LIN {X -190.795,Y +430.646,Z +0.000,A +0.152,E1 -46.707,E3 +41715.361,E4 +0.000} C_DIS
LIN {X -190.395,Y +441.145,Z +0.000,A +0.001,E1 -46.583,E3 +41728.754,E4 +0.000} C_DIS
LIN {X -190.239,Y +451.150,Z +0.000,A -0.000,E1 -46.528,E3 +41741.522,E4 +0.000} C_DIS
LIN {X -190.161,Y +465.026,Z +0.000,A -0.000,E1 -46.506,E3 +41759.237,E4 +0.000} C_DIS
LIN {X -190.142,Y +1057.148,Z +0.000,A -0.000,E1 -46.500,E3 +42515.443,E4 +0.000} C_DIS
LIN {X -190.147,Y +1068.924,Z +0.000,A -0.000,E1 -46.499,E3 +42530.484,E4 +0.000} C_DIS
LIN {X -190.159,Y +1079.072,Z +0.000,A -0.000,E1 -46.493,E3 +42543.449,E4 +0.000} C_DIS
LIN {X -190.174,Y +1086.028,Z +0.000,A -0.000,E1 -46.483,E3 +42552.343,E4 +0.000} C_DIS
LIN {X -190.200,Y +1096.186,Z +0.000,A -0.000,E1 -46.448,E3 +42565.347,E4 +0.000} C_DIS
LIN {X -190.154,Y +1108.998,Z +0.000,A -0.054,E1 -46.295,E3 +42581.842,E4 +0.000} C_DIS
LIN {X -189.772,Y +1119.341,Z +0.000,A -0.752,E1 -45.902,E3 +42595.380,E4 +0.000} C_DIS
LIN {X -189.097,Y +1124.276,Z +0.000,A -2.508,E1 -45.397,E3 +42602.112,E4 +0.000} C_DIS
LIN {X -187.410,Y +1129.069,Z +0.000,A -5.304,E1 -44.585,E3 +42609.285,E4 +0.000} C_DIS
LIN {X -183.899,Y +1134.873,Z +0.000,A -10.372,E1 -42.805,E3 +42619.291,E4 +0.000} C_DIS
LIN {X -179.711,Y +1140.065,Z +0.000,A -15.940,E1 -40.393,E3 +42630.077,E4 +0.000} C_DIS
LIN {X -176.763,Y +1143.197,Z +0.000,A -18.748,E1 -38.674,E3 +42637.815,E4 +0.000} C_DIS
LIN {X -172.185,Y +1147.423,Z +0.000,A -19.971,E1 -36.175,E3 +42650.545,E4 +0.000} C_DIS
LIN {X -165.999,Y +1152.127,Z +0.000,A -20.000,E1 -32.027,E3 +42670.303,E4 +0.000} C_DIS
LIN {X -160.138,Y +1155.667,Z +0.000,A -20.000,E1 -26.368,E3 +42694.673,E4 +0.000} C_DIS
LIN {X -155.625,Y +1157.756,Z +0.000,A -20.000,E1 -19.505,E3 +42723.349,E4 +0.000} C_DIS
LIN {X -153.552,Y +1158.113,Z +0.000,A -20.000,E1 -11.113,E3 +42759.100,E4 +0.000} C_DIS
LIN {X -156.311,Y +1155.540,Z +0.000,A -20.000,E1 -0.839,E3 +42802.460,E4 +0.000} C_DIS
LIN {X -161.281,Y +1151.851,Z +0.000,A -20.000,E1 +7.737,E3 +42832.359,E4 +0.000} C_DIS
LIN {X -167.493,Y +1147.157,Z +0.000,A -20.000,E1 +16.195,E3 +42856.798,E4 +0.000} C_DIS
LIN {X -173.235,Y +1142.221,Z +0.000,A -20.000,E1 +22.930,E3 +42874.100,E4 +0.000} C_DIS
LIN {X -181.123,Y +1133.734,Z +0.000,A -20.000,E1 +30.868,E3 +42894.856,E4 +0.000} C_DIS
LIN {X -189.654,Y +1120.856,Z +0.000,A -20.000,E1 +39.018,E3 +42916.870,E4 +0.000} C_DIS
LIN {X -195.246,Y +1107.046,Z +0.000,A -20.000,E1 +44.515,E3 +42934.772,E4 +0.000} C_DIS
LIN {X -198.051,Y +1092.368,Z +0.000,A -20.000,E1 +47.947,E3 +42951.298,E4 +0.000} C_DIS
LIN {X -198.143,Y +1081.370,Z +0.000,A -19.806,E1 +49.153,E3 +42963.159,E4 +0.000} C_DIS
LIN {X -197.177,Y +1073.569,Z +0.000,A -17.356,E1 +49.162,E3 +42971.743,E4 +0.000} C_DIS
LIN {X -195.448,Y +1066.139,Z +0.000,A -12.154,E1 +48.512,E3 +42980.338,E4 +0.000} C_DIS
LIN {X -193.346,Y +1058.941,Z +0.000,A -7.133,E1 +47.724,E3 +42989.218,E4 +0.000} C_DIS
LIN {X -191.781,Y +1050.839,Z +0.000,A -3.715,E1 +47.274,E3 +42999.551,E4 +0.000} C_DIS
LIN {X -190.795,Y +1039.355,Z +0.000,A -0.983,E1 +46.842,E3 +43014.211,E4 +0.000} C_DIS
LIN {X -190.395,Y +1028.856,Z +0.000,A -0.089,E1 +46.598,E3 +43027.605,E4 +0.000} C_DIS
LIN {X -190.239,Y +1018.851,Z +0.000,A -0.004,E1 +46.529,E3 +43040.373,E4 +0.000} C_DIS
LIN {X -190.161,Y +1004.975,Z +0.000,A +0.000,E1 +46.506,E3 +43058.087,E4 +0.000} C_DIS
LIN {X -190.142,Y +412.853,Z +0.000,A +0.000,E1 +46.501,E3 +43814.293,E4 +0.000} C_DIS
LIN {X -190.147,Y +401.077,Z +0.000,A +0.000,E1 +46.499,E3 +43829.334,E4 +0.000} C_DIS
LIN {X -190.159,Y +390.929,Z +0.000,A +0.000,E1 +46.494,E3 +43842.300,E4 +0.000} C_DIS
LIN {X -190.174,Y +383.973,Z +0.000,A +0.000,E1 +46.484,E3 +43851.193,E4 +0.000} C_DIS
LIN {X -190.200,Y +373.815,Z +0.000,A +0.000,E1 +46.448,E3 +43864.198,E4 +0.000} C_DIS
LIN {X -190.154,Y +361.003,Z +0.000,A +0.000,E1 +46.303,E3 +43880.692,E4 +0.000} C_DIS
LIN {X -189.772,Y +350.660,Z +0.000,A +0.049,E1 +45.996,E3 +43894.231,E4 +0.000} C_DIS
LIN {X -189.325,Y +346.917,Z +0.000,A +0.243,E1 +45.771,E3 +43899.300,E4 +0.000} C_DIS
LIN {X -188.196,Y +342.754,Z +0.000,A +1.966,E1 +45.249,E3 +43905.308,E4 +0.000} C_DIS
LIN {X -185.199,Y +337.023,Z +0.000,A +6.630,E1 +43.793,E3 +43914.682,E4 +0.000} C_DIS
LIN {X -181.141,Y +331.596,Z +0.000,A +12.274,E1 +41.569,E3 +43925.242,E4 +0.000} C_DIS
LIN {X -176.762,Y +326.804,Z +0.000,A +17.560,E1 +38.898,E3 +43936.666,E4 +0.000} C_DIS
LIN {X -172.184,Y +322.578,Z +0.000,A +19.859,E1 +36.197,E3 +43949.396,E4 +0.000} C_DIS
LIN {X -165.998,Y +317.874,Z +0.000,A +20.000,E1 +32.027,E3 +43969.154,E4 +0.000} C_DIS
LIN {X -160.137,Y +314.334,Z +0.000,A +20.000,E1 +26.368,E3 +43993.523,E4 +0.000} C_DIS
LIN {X -155.624,Y +312.245,Z +0.000,A +20.000,E1 +19.506,E3 +44022.199,E4 +0.000} C_DIS
LIN {X -153.557,Y +311.879,Z +0.000,A +20.000,E1 +11.113,E3 +44057.954,E4 +0.000} C_DIS
LIN {X -155.320,Y +313.348,Z +0.000,A +20.000,E1 +3.401,E3 +44091.138,E4 +0.000} C_DIS
LIN {X -160.005,Y +315.804,Z +0.000,A +20.000,E1 -4.720,E3 +44121.516,E4 +0.000} C_DIS
LIN {X -164.504,Y +318.255,Z +0.000,A +20.000,E1 -10.663,E3 +44140.885,E4 +0.000} C_DIS
LIN {X -170.340,Y +322.684,Z +0.000,A +20.000,E1 -17.457,E3 +44160.917,E4 +0.000} C_DIS
LIN {X -175.568,Y +329.106,Z +0.000,A +20.000,E1 -24.747,E3 +44178.151,E4 +0.000} C_DIS
LIN {X -184.074,Y +340.065,Z +0.000,A +20.000,E1 -33.664,E3 +44201.091,E4 +0.000} C_DIS
LIN {X -190.779,Y +351.388,Z +0.000,A +20.000,E1 -40.083,E3 +44218.869,E4 +0.000} C_DIS
LIN {X -195.254,Y +362.955,Z +0.000,A +20.000,E1 -44.515,E3 +44233.622,E4 +0.000} C_DIS
LIN {X -197.754,Y +374.780,Z +0.000,A +20.000,E1 -47.450,E3 +44247.044,E4 +0.000} C_DIS
LIN {X -198.310,Y +383.215,Z +0.000,A +19.956,E1 -48.698,E3 +44256.168,E4 +0.000} C_DIS
LIN {X -197.912,Y +391.275,Z +0.000,A +18.601,E1 -49.158,E3 +44264.886,E4 +0.000} C_DIS
LIN {X -196.679,Y +398.944,Z +0.000,A +13.989,E1 -48.784,E3 +44273.440,E4 +0.000} C_DIS
LIN {X -194.742,Y +406.288,Z +0.000,A +8.476,E1 -48.001,E3 +44282.123,E4 +0.000} C_DIS
LIN {X -192.748,Y +413.472,Z +0.000,A +3.905,E1 -47.267,E3 +44291.133,E4 +0.000} C_DIS
LIN {X -191.781,Y +419.162,Z +0.000,A +1.739,E1 -46.975,E3 +44298.401,E4 +0.000} C_DIS
LIN {X -190.795,Y +430.646,Z +0.000,A +0.152,E1 -46.707,E3 +44313.062,E4 +0.000} C_DIS
LIN {X -190.395,Y +441.145,Z +0.000,A +0.001,E1 -46.583,E3 +44326.455,E4 +0.000} C_DIS
LIN {X -190.239,Y +451.150,Z +0.000,A -0.000,E1 -46.528,E3 +44339.223,E4 +0.000} C_DIS
LIN {X -190.161,Y +465.026,Z +0.000,A -0.000,E1 -46.506,E3 +44356.938,E4 +0.000} C_DIS
LIN {X -190.142,Y +1057.148,Z +0.000,A -0.000,E1 -46.500,E3 +45113.144,E4 +0.000} C_DIS
LIN {X -190.147,Y +1068.924,Z +0.000,A -0.000,E1 -46.499,E3 +45128.185,E4 +0.000} C_DIS
LIN {X -190.159,Y +1079.072,Z +0.000,A -0.000,E1 -46.493,E3 +45141.150,E4 +0.000} C_DIS
LIN {X -190.174,Y +1086.028,Z +0.000,A -0.000,E1 -46.483,E3 +45150.044,E4 +0.000} C_DIS
LIN {X -190.200,Y +1096.186,Z +0.000,A -0.000,E1 -46.448,E3 +45163.048,E4 +0.000} C_DIS
LIN {X -190.154,Y +1108.998,Z +0.000,A -0.054,E1 -46.295,E3 +45179.543,E4 +0.000} C_DIS
LIN {X -189.772,Y +1119.341,Z +0.000,A -0.752,E1 -45.902,E3 +45193.081,E4 +0.000} C_DIS
LIN {X -189.097,Y +1124.276,Z +0.000,A -2.508,E1 -45.397,E3 +45199.813,E4 +0.000} C_DIS
LIN {X -187.410,Y +1129.069,Z +0.000,A -5.304,E1 -44.585,E3 +45206.986,E4 +0.000} C_DIS
LIN {X -183.899,Y +1134.873,Z +0.000,A -10.372,E1 -42.805,E3 +45216.992,E4 +0.000} C_DIS
LIN {X -179.711,Y +1140.065,Z +0.000,A -15.940,E1 -40.393,E3 +45227.778,E4 +0.000} C_DIS
LIN {X -176.763,Y +1143.197,Z +0.000,A -18.748,E1 -38.674,E3 +45235.516,E4 +0.000} C_DIS
LIN {X -172.185,Y +1147.423,Z +0.000,A -19.971,E1 -36.175,E3 +45248.246,E4 +0.000} C_DIS
LIN {X -165.999,Y +1152.127,Z +0.000,A -20.000,E1 -32.027,E3 +45268.004,E4 +0.000} C_DIS
LIN {X -160.138,Y +1155.667,Z +0.000,A -20.000,E1 -26.368,E3 +45292.374,E4 +0.000} C_DIS
LIN {X -155.625,Y +1157.756,Z +0.000,A -20.000,E1 -19.505,E3 +45321.050,E4 +0.000} C_DIS
LIN {X -153.552,Y +1158.113,Z +0.000,A -20.000,E1 -11.113,E3 +45356.801,E4 +0.000} C_DIS
LIN {X -156.311,Y +1155.540,Z +0.000,A -20.000,E1 -0.839,E3 +45400.161,E4 +0.000} C_DIS
LIN {X -161.281,Y +1151.851,Z +0.000,A -20.000,E1 +7.737,E3 +45430.060,E4 +0.000} C_DIS
LIN {X -167.493,Y +1147.157,Z +0.000,A -20.000,E1 +16.195,E3 +45454.499,E4 +0.000} C_DIS
LIN {X -173.235,Y +1142.221,Z +0.000,A -20.000,E1 +22.930,E3 +45471.801,E4 +0.000} C_DIS
LIN {X -181.123,Y +1133.734,Z +0.000,A -20.000,E1 +30.868,E3 +45492.557,E4 +0.000} C_DIS
LIN {X -189.654,Y +1120.856,Z +0.000,A -20.000,E1 +39.018,E3 +45514.571,E4 +0.000} C_DIS
LIN {X -195.246,Y +1107.046,Z +0.000,A -20.000,E1 +44.515,E3 +45532.473,E4 +0.000} C_DIS
LIN {X -198.051,Y +1092.368,Z +0.000,A -20.000,E1 +47.947,E3 +45548.999,E4 +0.000} C_DIS
LIN {X -198.143,Y +1081.370,Z +0.000,A -19.806,E1 +49.153,E3 +45560.860,E4 +0.000} C_DIS
LIN {X -197.177,Y +1073.569,Z +0.000,A -17.356,E1 +49.162,E3 +45569.444,E4 +0.000} C_DIS
LIN {X -195.448,Y +1066.139,Z +0.000,A -12.154,E1 +48.512,E3 +45578.039,E4 +0.000} C_DIS
LIN {X -193.346,Y +1058.941,Z +0.000,A -7.133,E1 +47.724,E3 +45586.919,E4 +0.000} C_DIS
LIN {X -191.781,Y +1050.839,Z +0.000,A -3.715,E1 +47.274,E3 +45597.252,E4 +0.000} C_DIS
LIN {X -190.795,Y +1039.355,Z +0.000,A -0.983,E1 +46.842,E3 +45611.912,E4 +0.000} C_DIS
LIN {X -190.395,Y +1028.856,Z +0.000,A -0.089,E1 +46.598,E3 +45625.306,E4 +0.000} C_DIS
LIN {X -190.239,Y +1018.851,Z +0.000,A -0.004,E1 +46.529,E3 +45638.074,E4 +0.000} C_DIS
LIN {X -190.161,Y +1004.975,Z +0.000,A +0.000,E1 +46.506,E3 +45655.788,E4 +0.000} C_DIS
LIN {X -190.142,Y +412.853,Z +0.000,A +0.000,E1 +46.501,E3 +46411.994,E4 +0.000} C_DIS
LIN {X -190.147,Y +401.077,Z +0.000,A +0.000,E1 +46.499,E3 +46427.035,E4 +0.000} C_DIS
LIN {X -190.159,Y +390.929,Z +0.000,A +0.000,E1 +46.494,E3 +46440.001,E4 +0.000} C_DIS
LIN {X -190.174,Y +383.973,Z +0.000,A +0.000,E1 +46.484,E3 +46448.894,E4 +0.000} C_DIS
LIN {X -190.200,Y +373.815,Z +0.000,A +0.000,E1 +46.448,E3 +46461.899,E4 +0.000} C_DIS
LIN {X -190.154,Y +361.003,Z +0.000,A +0.000,E1 +46.303,E3 +46478.393,E4 +0.000} C_DIS
LIN {X -189.772,Y +350.660,Z +0.000,A +0.049,E1 +45.996,E3 +46491.932,E4 +0.000} C_DIS
LIN {X -189.325,Y +346.917,Z +0.000,A +0.243,E1 +45.771,E3 +46497.001,E4 +0.000} C_DIS
LIN {X -188.196,Y +342.754,Z +0.000,A +1.966,E1 +45.249,E3 +46503.009,E4 +0.000} C_DIS
LIN {X -185.199,Y +337.023,Z +0.000,A +6.630,E1 +43.793,E3 +46512.383,E4 +0.000} C_DIS
LIN {X -181.141,Y +331.596,Z +0.000,A +12.274,E1 +41.569,E3 +46522.943,E4 +0.000} C_DIS
LIN {X -176.762,Y +326.804,Z +0.000,A +17.560,E1 +38.898,E3 +46534.367,E4 +0.000} C_DIS
LIN {X -172.184,Y +322.578,Z +0.000,A +19.859,E1 +36.197,E3 +46547.097,E4 +0.000} C_DIS
LIN {X -165.998,Y +317.874,Z +0.000,A +20.000,E1 +32.027,E3 +46566.855,E4 +0.000} C_DIS
LIN {X -160.137,Y +314.334,Z +0.000,A +20.000,E1 +26.368,E3 +46591.224,E4 +0.000} C_DIS
LIN {X -155.624,Y +312.245,Z +0.000,A +20.000,E1 +19.506,E3 +46619.900,E4 +0.000} C_DIS
LIN {X -153.557,Y +311.879,Z +0.000,A +20.000,E1 +11.113,E3 +46655.655,E4 +0.000} C_DIS
LIN {X -155.320,Y +313.348,Z +0.000,A +20.000,E1 +3.401,E3 +46688.839,E4 +0.000} C_DIS
LIN {X -160.005,Y +315.804,Z +0.000,A +20.000,E1 -4.720,E3 +46719.217,E4 +0.000} C_DIS
LIN {X -164.504,Y +318.255,Z +0.000,A +20.000,E1 -10.663,E3 +46738.586,E4 +0.000} C_DIS
LIN {X -170.340,Y +322.684,Z +0.000,A +20.000,E1 -17.457,E3 +46758.618,E4 +0.000} C_DIS
LIN {X -175.568,Y +329.106,Z +0.000,A +20.000,E1 -24.747,E3 +46775.852,E4 +0.000} C_DIS
LIN {X -184.074,Y +340.065,Z +0.000,A +20.000,E1 -33.664,E3 +46798.792,E4 +0.000} C_DIS
LIN {X -190.779,Y +351.388,Z +0.000,A +20.000,E1 -40.083,E3 +46816.570,E4 +0.000} C_DIS
LIN {X -195.254,Y +362.955,Z +0.000,A +20.000,E1 -44.515,E3 +46831.323,E4 +0.000} C_DIS
LIN {X -197.754,Y +374.780,Z +0.000,A +20.000,E1 -47.450,E3 +46844.745,E4 +0.000} C_DIS
LIN {X -198.310,Y +383.215,Z +0.000,A +19.956,E1 -48.698,E3 +46853.869,E4 +0.000} C_DIS
LIN {X -197.912,Y +391.275,Z +0.000,A +18.601,E1 -49.158,E3 +46862.587,E4 +0.000} C_DIS
LIN {X -196.679,Y +398.944,Z +0.000,A +13.989,E1 -48.784,E3 +46871.141,E4 +0.000} C_DIS
LIN {X -194.742,Y +406.288,Z +0.000,A +8.476,E1 -48.001,E3 +46879.824,E4 +0.000} C_DIS
LIN {X -192.748,Y +413.472,Z +0.000,A +3.905,E1 -47.267,E3 +46888.834,E4 +0.000} C_DIS
LIN {X -191.781,Y +419.162,Z +0.000,A +1.739,E1 -46.975,E3 +46896.102,E4 +0.000} C_DIS
LIN {X -190.795,Y +430.646,Z +0.000,A +0.152,E1 -46.707,E3 +46910.763,E4 +0.000} C_DIS
LIN {X -190.395,Y +441.145,Z +0.000,A +0.001,E1 -46.583,E3 +46924.156,E4 +0.000} C_DIS
LIN {X -190.239,Y +451.150,Z +0.000,A -0.000,E1 -46.528,E3 +46936.924,E4 +0.000} C_DIS
LIN {X -190.161,Y +465.026,Z +0.000,A -0.000,E1 -46.506,E3 +46954.639,E4 +0.000} C_DIS
LIN {X -190.142,Y +1057.148,Z +0.000,A -0.000,E1 -46.500,E3 +47710.845,E4 +0.000} C_DIS
LIN {X -190.147,Y +1068.924,Z +0.000,A -0.000,E1 -46.499,E3 +47725.886,E4 +0.000} C_DIS
LIN {X -190.159,Y +1079.072,Z +0.000,A -0.000,E1 -46.493,E3 +47738.851,E4 +0.000} C_DIS
LIN {X -190.174,Y +1086.028,Z +0.000,A -0.000,E1 -46.483,E3 +47747.745,E4 +0.000} C_DIS
LIN {X -190.200,Y +1096.186,Z +0.000,A -0.000,E1 -46.448,E3 +47760.749,E4 +0.000} C_DIS
LIN {X -190.154,Y +1108.998,Z +0.000,A -0.054,E1 -46.295,E3 +47777.244,E4 +0.000} C_DIS
LIN {X -189.772,Y +1119.341,Z +0.000,A -0.752,E1 -45.902,E3 +47790.782,E4 +0.000} C_DIS
LIN {X -189.097,Y +1124.276,Z +0.000,A -2.508,E1 -45.397,E3 +47797.514,E4 +0.000} C_DIS
LIN {X -187.410,Y +1129.069,Z +0.000,A -5.304,E1 -44.585,E3 +47804.687,E4 +0.000} C_DIS
LIN {X -183.899,Y +1134.873,Z +0.000,A -10.372,E1 -42.805,E3 +47814.693,E4 +0.000} C_DIS
LIN {X -179.711,Y +1140.065,Z +0.000,A -15.940,E1 -40.393,E3 +47825.479,E4 +0.000} C_DIS
LIN {X -176.763,Y +1143.197,Z +0.000,A -18.748,E1 -38.674,E3 +47833.217,E4 +0.000} C_DIS
LIN {X -172.185,Y +1147.423,Z +0.000,A -19.971,E1 -36.175,E3 +47845.947,E4 +0.000} C_DIS
LIN {X -165.999,Y +1152.127,Z +0.000,A -20.000,E1 -32.027,E3 +47865.705,E4 +0.000} C_DIS
LIN {X -160.138,Y +1155.667,Z +0.000,A -20.000,E1 -26.368,E3 +47890.075,E4 +0.000} C_DIS
LIN {X -155.625,Y +1157.756,Z +0.000,A -20.000,E1 -19.505,E3 +47918.751,E4 +0.000} C_DIS
LIN {X -153.552,Y +1158.113,Z +0.000,A -20.000,E1 -11.113,E3 +47954.502,E4 +0.000} C_DIS
LIN {X -156.311,Y +1155.540,Z +0.000,A -20.000,E1 -0.839,E3 +47997.862,E4 +0.000} C_DIS
LIN {X -161.281,Y +1151.851,Z +0.000,A -20.000,E1 +7.737,E3 +48027.761,E4 +0.000} C_DIS
LIN {X -167.493,Y +1147.157,Z +0.000,A -20.000,E1 +16.195,E3 +48052.200,E4 +0.000} C_DIS
LIN {X -173.235,Y +1142.221,Z +0.000,A -20.000,E1 +22.930,E3 +48069.502,E4 +0.000} C_DIS
LIN {X -181.123,Y +1133.734,Z +0.000,A -20.000,E1 +30.868,E3 +48090.258,E4 +0.000} C_DIS
LIN {X -189.654,Y +1120.856,Z +0.000,A -20.000,E1 +39.018,E3 +48112.272,E4 +0.000} C_DIS
LIN {X -195.246,Y +1107.046,Z +0.000,A -20.000,E1 +44.515,E3 +48130.174,E4 +0.000} C_DIS
LIN {X -198.051,Y +1092.368,Z +0.000,A -20.000,E1 +47.947,E3 +48146.700,E4 +0.000} C_DIS
LIN {X -198.143,Y +1081.370,Z +0.000,A -19.806,E1 +49.153,E3 +48158.561,E4 +0.000} C_DIS
LIN {X -197.177,Y +1073.569,Z +0.000,A -17.356,E1 +49.162,E3 +48167.145,E4 +0.000} C_DIS
LIN {X -195.448,Y +1066.139,Z +0.000,A -12.154,E1 +48.512,E3 +48175.740,E4 +0.000} C_DIS
LIN {X -193.346,Y +1058.941,Z +0.000,A -7.133,E1 +47.724,E3 +48184.620,E4 +0.000} C_DIS
LIN {X -191.781,Y +1050.839,Z +0.000,A -3.715,E1 +47.274,E3 +48194.953,E4 +0.000} C_DIS
LIN {X -190.795,Y +1039.355,Z +0.000,A -0.983,E1 +46.842,E3 +48209.613,E4 +0.000} C_DIS
LIN {X -190.395,Y +1028.856,Z +0.000,A -0.089,E1 +46.598,E3 +48223.007,E4 +0.000} C_DIS
LIN {X -190.239,Y +1018.851,Z +0.000,A -0.004,E1 +46.529,E3 +48235.775,E4 +0.000} C_DIS
LIN {X -190.161,Y +1004.975,Z +0.000,A +0.000,E1 +46.506,E3 +48253.489,E4 +0.000} C_DIS
LIN {X -190.142,Y +412.853,Z +0.000,A +0.000,E1 +46.501,E3 +49009.695,E4 +0.000} C_DIS
LIN {X -190.147,Y +401.077,Z +0.000,A +0.000,E1 +46.499,E3 +49024.736,E4 +0.000} C_DIS
LIN {X -190.159,Y +390.929,Z +0.000,A +0.000,E1 +46.494,E3 +49037.702,E4 +0.000} C_DIS
LIN {X -190.174,Y +383.973,Z +0.000,A +0.000,E1 +46.484,E3 +49046.595,E4 +0.000} C_DIS
LIN {X -190.200,Y +373.815,Z +0.000,A +0.000,E1 +46.448,E3 +49059.600,E4 +0.000} C_DIS
LIN {X -190.154,Y +361.003,Z +0.000,A +0.000,E1 +46.303,E3 +49076.094,E4 +0.000} C_DIS
LIN {X -189.772,Y +350.660,Z +0.000,A +0.049,E1 +45.996,E3 +49089.633,E4 +0.000} C_DIS
LIN {X -189.325,Y +346.917,Z +0.000,A +0.243,E1 +45.771,E3 +49094.702,E4 +0.000} C_DIS
LIN {X -188.196,Y +342.754,Z +0.000,A +1.966,E1 +45.249,E3 +49100.710,E4 +0.000} C_DIS
LIN {X -185.199,Y +337.023,Z +0.000,A +6.630,E1 +43.793,E3 +49110.084,E4 +0.000} C_DIS
LIN {X -181.141,Y +331.596,Z +0.000,A +12.274,E1 +41.569,E3 +49120.644,E4 +0.000} C_DIS
LIN {X -176.762,Y +326.804,Z +0.000,A +17.560,E1 +38.898,E3 +49132.068,E4 +0.000} C_DIS
LIN {X -172.184,Y +322.578,Z +0.000,A +19.859,E1 +36.197,E3 +49144.798,E4 +0.000} C_DIS
LIN {X -165.998,Y +317.874,Z +0.000,A +20.000,E1 +32.027,E3 +49164.556,E4 +0.000} C_DIS
LIN {X -160.137,Y +314.334,Z +0.000,A +20.000,E1 +26.368,E3 +49188.925,E4 +0.000} C_DIS
LIN {X -155.624,Y +312.245,Z +0.000,A +20.000,E1 +19.506,E3 +49217.601,E4 +0.000} C_DIS
LIN {X -153.557,Y +311.879,Z +0.000,A +20.000,E1 +11.113,E3 +49253.356,E4 +0.000} C_DIS
LIN {X -155.320,Y +313.348,Z +0.000,A +20.000,E1 +3.401,E3 +49286.540,E4 +0.000} C_DIS
LIN {X -160.005,Y +315.804,Z +0.000,A +20.000,E1 -4.720,E3 +49316.918,E4 +0.000} C_DIS
LIN {X -164.504,Y +318.255,Z +0.000,A +20.000,E1 -10.663,E3 +49336.287,E4 +0.000} C_DIS
LIN {X -170.340,Y +322.684,Z +0.000,A +20.000,E1 -17.457,E3 +49356.319,E4 +0.000} C_DIS
LIN {X -175.568,Y +329.106,Z +0.000,A +20.000,E1 -24.747,E3 +49373.553,E4 +0.000} C_DIS
LIN {X -184.074,Y +340.065,Z +0.000,A +20.000,E1 -33.664,E3 +49396.493,E4 +0.000} C_DIS
LIN {X -190.779,Y +351.388,Z +0.000,A +20.000,E1 -40.083,E3 +49414.271,E4 +0.000} C_DIS
LIN {X -195.254,Y +362.955,Z +0.000,A +20.000,E1 -44.515,E3 +49429.024,E4 +0.000} C_DIS
LIN {X -197.754,Y +374.780,Z +0.000,A +20.000,E1 -47.450,E3 +49442.446,E4 +0.000} C_DIS
LIN {X -198.310,Y +383.215,Z +0.000,A +19.956,E1 -48.698,E3 +49451.570,E4 +0.000} C_DIS
LIN {X -197.912,Y +391.275,Z +0.000,A +18.601,E1 -49.158,E3 +49460.288,E4 +0.000} C_DIS
LIN {X -196.679,Y +398.944,Z +0.000,A +13.989,E1 -48.784,E3 +49468.842,E4 +0.000} C_DIS
LIN {X -194.742,Y +406.288,Z +0.000,A +8.476,E1 -48.001,E3 +49477.525,E4 +0.000} C_DIS
LIN {X -192.748,Y +413.472,Z +0.000,A +3.905,E1 -47.267,E3 +49486.535,E4 +0.000} C_DIS
LIN {X -191.781,Y +419.162,Z +0.000,A +1.739,E1 -46.975,E3 +49493.803,E4 +0.000} C_DIS
LIN {X -190.795,Y +430.646,Z +0.000,A +0.152,E1 -46.707,E3 +49508.464,E4 +0.000} C_DIS
LIN {X -190.395,Y +441.145,Z +0.000,A +0.001,E1 -46.583,E3 +49521.857,E4 +0.000} C_DIS
LIN {X -190.239,Y +451.150,Z +0.000,A -0.000,E1 -46.528,E3 +49534.625,E4 +0.000} C_DIS
LIN {X -190.161,Y +465.026,Z +0.000,A -0.000,E1 -46.506,E3 +49552.340,E4 +0.000} C_DIS
LIN {X -190.142,Y +1057.148,Z +0.000,A -0.000,E1 -46.500,E3 +50308.546,E4 +0.000} C_DIS
LIN {X -190.147,Y +1068.924,Z +0.000,A -0.000,E1 -46.499,E3 +50323.587,E4 +0.000} C_DIS
LIN {X -190.159,Y +1079.072,Z +0.000,A -0.000,E1 -46.493,E3 +50336.552,E4 +0.000} C_DIS
LIN {X -190.174,Y +1086.028,Z +0.000,A -0.000,E1 -46.483,E3 +50345.446,E4 +0.000} C_DIS
LIN {X -190.200,Y +1096.186,Z +0.000,A -0.000,E1 -46.448,E3 +50358.450,E4 +0.000} C_DIS
LIN {X -190.154,Y +1108.998,Z +0.000,A -0.054,E1 -46.295,E3 +50374.945,E4 +0.000} C_DIS
LIN {X -189.772,Y +1119.341,Z +0.000,A -0.752,E1 -45.902,E3 +50388.483,E4 +0.000} C_DIS
LIN {X -189.097,Y +1124.276,Z +0.000,A -2.508,E1 -45.397,E3 +50395.215,E4 +0.000} C_DIS
LIN {X -187.410,Y +1129.069,Z +0.000,A -5.304,E1 -44.585,E3 +50402.388,E4 +0.000} C_DIS
LIN {X -183.899,Y +1134.873,Z +0.000,A -10.372,E1 -42.805,E3 +50412.394,E4 +0.000} C_DIS
LIN {X -179.711,Y +1140.065,Z +0.000,A -15.940,E1 -40.393,E3 +50423.180,E4 +0.000} C_DIS
LIN {X -176.763,Y +1143.197,Z +0.000,A -18.748,E1 -38.674,E3 +50430.918,E4 +0.000} C_DIS
LIN {X -172.185,Y +1147.423,Z +0.000,A -19.971,E1 -36.175,E3 +50443.648,E4 +0.000} C_DIS
LIN {X -165.999,Y +1152.127,Z +0.000,A -20.000,E1 -32.027,E3 +50463.406,E4 +0.000} C_DIS
LIN {X -160.138,Y +1155.667,Z +0.000,A -20.000,E1 -26.368,E3 +50487.776,E4 +0.000} C_DIS
LIN {X -155.625,Y +1157.756,Z +0.000,A -20.000,E1 -19.505,E3 +50516.452,E4 +0.000} C_DIS
LIN {X -153.552,Y +1158.113,Z +0.000,A -20.000,E1 -11.113,E3 +50552.203,E4 +0.000} C_DIS
LIN {X -156.311,Y +1155.540,Z +0.000,A -20.000,E1 -0.839,E3 +50595.563,E4 +0.000} C_DIS
LIN {X -161.281,Y +1151.851,Z +0.000,A -20.000,E1 +7.737,E3 +50625.462,E4 +0.000} C_DIS
LIN {X -167.493,Y +1147.157,Z +0.000,A -20.000,E1 +16.195,E3 +50649.901,E4 +0.000} C_DIS
LIN {X -173.235,Y +1142.221,Z +0.000,A -20.000,E1 +22.930,E3 +50667.203,E4 +0.000} C_DIS
LIN {X -181.123,Y +1133.734,Z +0.000,A -20.000,E1 +30.868,E3 +50687.959,E4 +0.000} C_DIS
LIN {X -189.654,Y +1120.856,Z +0.000,A -20.000,E1 +39.018,E3 +50709.973,E4 +0.000} C_DIS
LIN {X -195.246,Y +1107.046,Z +0.000,A -20.000,E1 +44.515,E3 +50727.875,E4 +0.000} C_DIS
LIN {X -198.051,Y +1092.368,Z +0.000,A -20.000,E1 +47.947,E3 +50744.401,E4 +0.000} C_DIS
LIN {X -198.143,Y +1081.370,Z +0.000,A -19.806,E1 +49.153,E3 +50756.262,E4 +0.000} C_DIS
LIN {X -197.177,Y +1073.569,Z +0.000,A -17.356,E1 +49.162,E3 +50764.846,E4 +0.000} C_DIS
LIN {X -195.448,Y +1066.139,Z +0.000,A -12.154,E1 +48.512,E3 +50773.441,E4 +0.000} C_DIS
LIN {X -193.346,Y +1058.941,Z +0.000,A -7.133,E1 +47.724,E3 +50782.321,E4 +0.000} C_DIS
LIN {X -191.781,Y +1050.839,Z +0.000,A -3.715,E1 +47.274,E3 +50792.654,E4 +0.000} C_DIS
LIN {X -190.795,Y +1039.355,Z +0.000,A -0.983,E1 +46.842,E3 +50807.314,E4 +0.000} C_DIS
LIN {X -190.395,Y +1028.856,Z +0.000,A -0.089,E1 +46.598,E3 +50820.708,E4 +0.000} C_DIS
LIN {X -190.239,Y +1018.851,Z +0.000,A -0.004,E1 +46.529,E3 +50833.476,E4 +0.000} C_DIS
LIN {X -190.161,Y +1004.975,Z +0.000,A +0.000,E1 +46.506,E3 +50851.190,E4 +0.000} C_DIS
LIN {X -190.142,Y +412.853,Z +0.000,A +0.000,E1 +46.501,E3 +51607.396,E4 +0.000} C_DIS
LIN {X -190.147,Y +401.077,Z +0.000,A +0.000,E1 +46.499,E3 +51622.437,E4 +0.000} C_DIS
LIN {X -190.159,Y +390.929,Z +0.000,A +0.000,E1 +46.494,E3 +51635.403,E4 +0.000} C_DIS
LIN {X -190.174,Y +383.973,Z +0.000,A +0.000,E1 +46.484,E3 +51644.296,E4 +0.000} C_DIS
LIN {X -190.200,Y +373.815,Z +0.000,A +0.000,E1 +46.448,E3 +51657.301,E4 +0.000} C_DIS
LIN {X -190.154,Y +361.003,Z +0.000,A +0.000,E1 +46.303,E3 +51673.795,E4 +0.000} C_DIS
LIN {X -189.772,Y +350.660,Z +0.000,A +0.049,E1 +45.996,E3 +51687.334,E4 +0.000} C_DIS
LIN {X -189.325,Y +346.917,Z +0.000,A +0.243,E1 +45.771,E3 +51692.403,E4 +0.000} C_DIS
LIN {X -188.196,Y +342.754,Z +0.000,A +1.966,E1 +45.249,E3 +51698.411,E4 +0.000} C_DIS
LIN {X -185.199,Y +337.023,Z +0.000,A +6.630,E1 +43.793,E3 +51707.785,E4 +0.000} C_DIS
LIN {X -181.141,Y +331.596,Z +0.000,A +12.274,E1 +41.569,E3 +51718.345,E4 +0.000} C_DIS
LIN {X -176.762,Y +326.804,Z +0.000,A +17.560,E1 +38.898,E3 +51729.769,E4 +0.000} C_DIS
LIN {X -172.184,Y +322.578,Z +0.000,A +19.859,E1 +36.197,E3 +51742.499,E4 +0.000} C_DIS
LIN {X -165.998,Y +317.874,Z +0.000,A +20.000,E1 +32.027,E3 +51762.257,E4 +0.000} C_DIS
LIN {X -160.137,Y +314.334,Z +0.000,A +20.000,E1 +26.368,E3 +51786.626,E4 +0.000} C_DIS
LIN {X -155.624,Y +312.245,Z +0.000,A +20.000,E1 +19.506,E3 +51815.302,E4 +0.000} C_DIS
LIN {X -153.557,Y +311.879,Z +0.000,A +20.000,E1 +11.113,E3 +51851.057,E4 +0.000} C_DIS
LIN {X -155.320,Y +313.348,Z +0.000,A +20.000,E1 +3.401,E3 +51884.241,E4 +0.000} C_DIS
LIN {X -160.005,Y +315.804,Z +0.000,A +20.000,E1 -4.720,E3 +51914.619,E4 +0.000} C_DIS
LIN {X -164.504,Y +318.255,Z +0.000,A +20.000,E1 -10.663,E3 +51933.988,E4 +0.000} C_DIS
LIN {X -170.340,Y +322.684,Z +0.000,A +20.000,E1 -17.457,E3 +51954.020,E4 +0.000} C_DIS
LIN {X -175.568,Y +329.106,Z +0.000,A +20.000,E1 -24.747,E3 +51971.254,E4 +0.000} C_DIS
LIN {X -184.074,Y +340.065,Z +0.000,A +20.000,E1 -33.664,E3 +51994.194,E4 +0.000} C_DIS
LIN {X -190.779,Y +351.388,Z +0.000,A +20.000,E1 -40.083,E3 +52011.972,E4 +0.000} C_DIS
LIN {X -195.254,Y +362.955,Z +0.000,A +20.000,E1 -44.515,E3 +52026.725,E4 +0.000} C_DIS
LIN {X -197.754,Y +374.780,Z +0.000,A +20.000,E1 -47.450,E3 +52040.147,E4 +0.000} C_DIS
LIN {X -198.310,Y +383.215,Z +0.000,A +19.956,E1 -48.698,E3 +52049.271,E4 +0.000} C_DIS
LIN {X -197.912,Y +391.275,Z +0.000,A +18.601,E1 -49.158,E3 +52057.989,E4 +0.000} C_DIS
LIN {X -196.679,Y +398.944,Z +0.000,A +13.989,E1 -48.784,E3 +52066.543,E4 +0.000} C_DIS
LIN {X -194.742,Y +406.288,Z +0.000,A +8.476,E1 -48.001,E3 +52075.226,E4 +0.000} C_DIS
LIN {X -192.748,Y +413.472,Z +0.000,A +3.905,E1 -47.267,E3 +52084.236,E4 +0.000} C_DIS
LIN {X -191.781,Y +419.162,Z +0.000,A +1.739,E1 -46.975,E3 +52091.504,E4 +0.000} C_DIS
LIN {X -190.795,Y +430.646,Z +0.000,A +0.152,E1 -46.707,E3 +52106.165,E4 +0.000} C_DIS
LIN {X -190.395,Y +441.145,Z +0.000,A +0.001,E1 -46.583,E3 +52119.558,E4 +0.000} C_DIS
LIN {X -190.239,Y +451.150,Z +0.000,A -0.000,E1 -46.528,E3 +52132.326,E4 +0.000} C_DIS
LIN {X -190.161,Y +465.026,Z +0.000,A -0.000,E1 -46.506,E3 +52150.041,E4 +0.000} C_DIS
LIN {X -190.142,Y +1057.148,Z +0.000,A -0.000,E1 -46.500,E3 +52906.247,E4 +0.000} C_DIS
LIN {X -190.147,Y +1068.924,Z +0.000,A -0.000,E1 -46.499,E3 +52921.288,E4 +0.000} C_DIS
LIN {X -190.159,Y +1079.072,Z +0.000,A -0.000,E1 -46.493,E3 +52934.253,E4 +0.000} C_DIS
LIN {X -190.174,Y +1086.028,Z +0.000,A -0.000,E1 -46.483,E3 +52943.147,E4 +0.000} C_DIS
LIN {X -190.200,Y +1096.186,Z +0.000,A -0.000,E1 -46.448,E3 +52956.151,E4 +0.000} C_DIS
LIN {X -190.154,Y +1108.998,Z +0.000,A -0.054,E1 -46.295,E3 +52972.646,E4 +0.000} C_DIS
LIN {X -189.772,Y +1119.341,Z +0.000,A -0.752,E1 -45.902,E3 +52986.184,E4 +0.000} C_DIS
LIN {X -189.097,Y +1124.276,Z +0.000,A -2.508,E1 -45.397,E3 +52992.916,E4 +0.000} C_DIS
LIN {X -187.410,Y +1129.069,Z +0.000,A -5.304,E1 -44.585,E3 +53000.089,E4 +0.000} C_DIS
LIN {X -183.899,Y +1134.873,Z +0.000,A -10.372,E1 -42.805,E3 +53010.095,E4 +0.000} C_DIS
LIN {X -179.711,Y +1140.065,Z +0.000,A -15.940,E1 -40.393,E3 +53020.881,E4 +0.000} C_DIS
LIN {X -176.763,Y +1143.197,Z +0.000,A -18.748,E1 -38.674,E3 +53028.619,E4 +0.000} C_DIS
LIN {X -172.185,Y +1147.423,Z +0.000,A -19.971,E1 -36.175,E3 +53041.349,E4 +0.000} C_DIS
LIN {X -165.999,Y +1152.127,Z +0.000,A -20.000,E1 -32.027,E3 +53061.107,E4 +0.000} C_DIS
LIN {X -160.138,Y +1155.667,Z +0.000,A -20.000,E1 -26.368,E3 +53085.477,E4 +0.000} C_DIS
LIN {X -155.625,Y +1157.756,Z +0.000,A -20.000,E1 -19.505,E3 +53114.153,E4 +0.000} C_DIS
LIN {X -153.552,Y +1158.113,Z +0.000,A -20.000,E1 -11.113,E3 +53149.904,E4 +0.000} C_DIS
LIN {X -156.311,Y +1155.540,Z +0.000,A -20.000,E1 -0.839,E3 +53193.264,E4 +0.000} C_DIS
LIN {X -161.281,Y +1151.851,Z +0.000,A -20.000,E1 +7.737,E3 +53223.163,E4 +0.000} C_DIS
LIN {X -167.493,Y +1147.157,Z +0.000,A -20.000,E1 +16.195,E3 +53247.602,E4 +0.000} C_DIS
LIN {X -173.235,Y +1142.221,Z +0.000,A -20.000,E1 +22.930,E3 +53264.904,E4 +0.000} C_DIS
LIN {X -181.123,Y +1133.734,Z +0.000,A -20.000,E1 +30.868,E3 +53285.660,E4 +0.000} C_DIS
LIN {X -189.654,Y +1120.856,Z +0.000,A -20.000,E1 +39.018,E3 +53307.674,E4 +0.000} C_DIS
LIN {X -195.246,Y +1107.046,Z +0.000,A -20.000,E1 +44.515,E3 +53325.576,E4 +0.000} C_DIS
LIN {X -198.051,Y +1092.368,Z +0.000,A -20.000,E1 +47.947,E3 +53342.102,E4 +0.000} C_DIS
LIN {X -198.143,Y +1081.370,Z +0.000,A -19.806,E1 +49.153,E3 +53353.963,E4 +0.000} C_DIS
LIN {X -197.177,Y +1073.569,Z +0.000,A -17.356,E1 +49.162,E3 +53362.547,E4 +0.000} C_DIS
LIN {X -195.448,Y +1066.139,Z +0.000,A -12.154,E1 +48.512,E3 +53371.142,E4 +0.000} C_DIS
LIN {X -193.346,Y +1058.941,Z +0.000,A -7.133,E1 +47.724,E3 +53380.022,E4 +0.000} C_DIS
LIN {X -191.781,Y +1050.839,Z +0.000,A -3.715,E1 +47.274,E3 +53390.355,E4 +0.000} C_DIS
LIN {X -190.795,Y +1039.355,Z +0.000,A -0.983,E1 +46.842,E3 +53405.015,E4 +0.000} C_DIS
LIN {X -190.395,Y +1028.856,Z +0.000,A -0.089,E1 +46.598,E3 +53418.409,E4 +0.000} C_DIS
LIN {X -190.239,Y +1018.851,Z +0.000,A -0.004,E1 +46.529,E3 +53431.177,E4 +0.000} C_DIS
LIN {X -190.161,Y +1004.975,Z +0.000,A +0.000,E1 +46.506,E3 +53448.891,E4 +0.000} C_DIS
LIN {X -190.142,Y +412.853,Z +0.000,A +0.000,E1 +46.501,E3 +54205.097,E4 +0.000} C_DIS
LIN {X -190.147,Y +401.077,Z +0.000,A +0.000,E1 +46.499,E3 +54220.138,E4 +0.000} C_DIS
LIN {X -190.159,Y +390.929,Z +0.000,A +0.000,E1 +46.494,E3 +54233.104,E4 +0.000} C_DIS
LIN {X -190.174,Y +383.973,Z +0.000,A +0.000,E1 +46.484,E3 +54241.997,E4 +0.000} C_DIS
LIN {X -190.200,Y +373.815,Z +0.000,A +0.000,E1 +46.448,E3 +54255.002,E4 +0.000} C_DIS
LIN {X -190.154,Y +361.003,Z +0.000,A +0.000,E1 +46.303,E3 +54271.496,E4 +0.000} C_DIS
LIN {X -189.772,Y +350.660,Z +0.000,A +0.049,E1 +45.996,E3 +54285.035,E4 +0.000} C_DIS
LIN {X -189.325,Y +346.917,Z +0.000,A +0.243,E1 +45.771,E3 +54290.104,E4 +0.000} C_DIS
LIN {X -188.196,Y +342.754,Z +0.000,A +1.966,E1 +45.249,E3 +54296.112,E4 +0.000} C_DIS
LIN {X -185.199,Y +337.023,Z +0.000,A +6.630,E1 +43.793,E3 +54305.486,E4 +0.000} C_DIS
LIN {X -181.141,Y +331.596,Z +0.000,A +12.274,E1 +41.569,E3 +54316.046,E4 +0.000} C_DIS
LIN {X -176.762,Y +326.804,Z +0.000,A +17.560,E1 +38.898,E3 +54327.470,E4 +0.000} C_DIS
LIN {X -172.184,Y +322.578,Z +0.000,A +19.859,E1 +36.197,E3 +54340.200,E4 +0.000} C_DIS
LIN {X -165.998,Y +317.874,Z +0.000,A +20.000,E1 +32.027,E3 +54359.958,E4 +0.000} C_DIS
LIN {X -160.137,Y +314.334,Z +0.000,A +20.000,E1 +26.368,E3 +54384.327,E4 +0.000} C_DIS
LIN {X -155.624,Y +312.245,Z +0.000,A +20.000,E1 +19.506,E3 +54413.003,E4 +0.000} C_DIS
LIN {X -153.557,Y +311.879,Z +0.000,A +20.000,E1 +11.113,E3 +54448.758,E4 +0.000} C_DIS
LIN {X -155.320,Y +313.348,Z +0.000,A +20.000,E1 +3.401,E3 +54481.942,E4 +0.000} C_DIS
LIN {X -160.005,Y +315.804,Z +0.000,A +20.000,E1 -4.720,E3 +54512.320,E4 +0.000} C_DIS
LIN {X -164.504,Y +318.255,Z +0.000,A +20.000,E1 -10.663,E3 +54531.689,E4 +0.000} C_DIS
LIN {X -170.340,Y +322.684,Z +0.000,A +20.000,E1 -17.457,E3 +54551.721,E4 +0.000} C_DIS
LIN {X -175.568,Y +329.106,Z +0.000,A +20.000,E1 -24.747,E3 +54568.955,E4 +0.000} C_DIS
LIN {X -184.074,Y +340.065,Z +0.000,A +20.000,E1 -33.664,E3 +54591.895,E4 +0.000} C_DIS
LIN {X -190.779,Y +351.388,Z +0.000,A +20.000,E1 -40.083,E3 +54609.673,E4 +0.000} C_DIS
LIN {X -195.254,Y +362.955,Z +0.000,A +20.000,E1 -44.515,E3 +54624.426,E4 +0.000} C_DIS
LIN {X -197.754,Y +374.780,Z +0.000,A +20.000,E1 -47.450,E3 +54637.848,E4 +0.000} C_DIS
LIN {X -198.310,Y +383.215,Z +0.000,A +19.956,E1 -48.698,E3 +54646.972,E4 +0.000} C_DIS
LIN {X -197.912,Y +391.275,Z +0.000,A +18.601,E1 -49.158,E3 +54655.690,E4 +0.000} C_DIS
LIN {X -196.679,Y +398.944,Z +0.000,A +13.989,E1 -48.784,E3 +54664.244,E4 +0.000} C_DIS
LIN {X -194.742,Y +406.288,Z +0.000,A +8.476,E1 -48.001,E3 +54672.927,E4 +0.000} C_DIS
LIN {X -192.748,Y +413.472,Z +0.000,A +3.905,E1 -47.267,E3 +54681.937,E4 +0.000} C_DIS
LIN {X -191.781,Y +419.162,Z +0.000,A +1.739,E1 -46.975,E3 +54689.205,E4 +0.000} C_DIS
LIN {X -190.795,Y +430.646,Z +0.000,A +0.152,E1 -46.707,E3 +54703.866,E4 +0.000} C_DIS
LIN {X -190.395,Y +441.145,Z +0.000,A +0.001,E1 -46.583,E3 +54717.259,E4 +0.000} C_DIS
LIN {X -190.239,Y +451.150,Z +0.000,A -0.000,E1 -46.528,E3 +54730.027,E4 +0.000} C_DIS
LIN {X -190.161,Y +465.026,Z +0.000,A -0.000,E1 -46.506,E3 +54747.742,E4 +0.000} C_DIS
LIN {X -190.142,Y +1057.148,Z +0.000,A -0.000,E1 -46.500,E3 +55503.948,E4 +0.000} C_DIS
LIN {X -190.147,Y +1068.924,Z +0.000,A -0.000,E1 -46.499,E3 +55518.989,E4 +0.000} C_DIS
LIN {X -190.159,Y +1079.072,Z +0.000,A -0.000,E1 -46.493,E3 +55531.954,E4 +0.000} C_DIS
LIN {X -190.174,Y +1086.028,Z +0.000,A -0.000,E1 -46.483,E3 +55540.848,E4 +0.000} C_DIS
LIN {X -190.200,Y +1096.186,Z +0.000,A -0.000,E1 -46.448,E3 +55553.852,E4 +0.000} C_DIS
LIN {X -190.154,Y +1108.998,Z +0.000,A -0.054,E1 -46.295,E3 +55570.347,E4 +0.000} C_DIS
LIN {X -189.772,Y +1119.341,Z +0.000,A -0.752,E1 -45.902,E3 +55583.885,E4 +0.000} C_DIS
LIN {X -189.097,Y +1124.276,Z +0.000,A -2.508,E1 -45.397,E3 +55590.617,E4 +0.000} C_DIS
LIN {X -187.410,Y +1129.069,Z +0.000,A -5.304,E1 -44.585,E3 +55597.790,E4 +0.000} C_DIS
LIN {X -183.899,Y +1134.873,Z +0.000,A -10.372,E1 -42.805,E3 +55607.796,E4 +0.000} C_DIS
LIN {X -179.711,Y +1140.065,Z +0.000,A -15.940,E1 -40.393,E3 +55618.582,E4 +0.000} C_DIS
LIN {X -176.763,Y +1143.197,Z +0.000,A -18.748,E1 -38.674,E3 +55626.320,E4 +0.000} C_DIS
LIN {X -172.185,Y +1147.423,Z +0.000,A -19.971,E1 -36.175,E3 +55639.050,E4 +0.000} C_DIS
LIN {X -165.999,Y +1152.127,Z +0.000,A -20.000,E1 -32.027,E3 +55658.808,E4 +0.000} C_DIS
LIN {X -160.138,Y +1155.667,Z +0.000,A -20.000,E1 -26.368,E3 +55683.178,E4 +0.000} C_DIS
LIN {X -155.625,Y +1157.756,Z +0.000,A -20.000,E1 -19.505,E3 +55711.854,E4 +0.000} C_DIS
LIN {X -153.552,Y +1158.113,Z +0.000,A -20.000,E1 -11.113,E3 +55747.605,E4 +0.000} C_DIS
LIN {X -156.311,Y +1155.540,Z +0.000,A -20.000,E1 -0.839,E3 +55790.965,E4 +0.000} C_DIS
LIN {X -161.281,Y +1151.851,Z +0.000,A -20.000,E1 +7.737,E3 +55820.864,E4 +0.000} C_DIS
LIN {X -167.493,Y +1147.157,Z +0.000,A -20.000,E1 +16.195,E3 +55845.303,E4 +0.000} C_DIS
LIN {X -173.235,Y +1142.221,Z +0.000,A -20.000,E1 +22.930,E3 +55862.605,E4 +0.000} C_DIS
LIN {X -181.123,Y +1133.734,Z +0.000,A -20.000,E1 +30.868,E3 +55883.361,E4 +0.000} C_DIS
LIN {X -189.654,Y +1120.856,Z +0.000,A -20.000,E1 +39.018,E3 +55905.375,E4 +0.000} C_DIS
LIN {X -195.246,Y +1107.046,Z +0.000,A -20.000,E1 +44.515,E3 +55923.277,E4 +0.000} C_DIS
LIN {X -198.051,Y +1092.368,Z +0.000,A -20.000,E1 +47.947,E3 +55939.803,E4 +0.000} C_DIS
LIN {X -198.143,Y +1081.370,Z +0.000,A -19.806,E1 +49.153,E3 +55951.664,E4 +0.000} C_DIS
LIN {X -197.177,Y +1073.569,Z +0.000,A -17.356,E1 +49.162,E3 +55960.248,E4 +0.000} C_DIS
LIN {X -195.448,Y +1066.139,Z +0.000,A -12.154,E1 +48.512,E3 +55968.843,E4 +0.000} C_DIS
LIN {X -193.346,Y +1058.941,Z +0.000,A -7.133,E1 +47.724,E3 +55977.723,E4 +0.000} C_DIS
LIN {X -191.781,Y +1050.839,Z +0.000,A -3.715,E1 +47.274,E3 +55988.056,E4 +0.000} C_DIS
LIN {X -190.795,Y +1039.355,Z +0.000,A -0.983,E1 +46.842,E3 +56002.716,E4 +0.000} C_DIS
LIN {X -190.395,Y +1028.856,Z +0.000,A -0.089,E1 +46.598,E3 +56016.110,E4 +0.000} C_DIS
LIN {X -190.239,Y +1018.851,Z +0.000,A -0.004,E1 +46.529,E3 +56028.878,E4 +0.000} C_DIS
LIN {X -190.161,Y +1004.975,Z +0.000,A +0.000,E1 +46.506,E3 +56046.592,E4 +0.000} C_DIS
LIN {X -190.142,Y +412.853,Z +0.000,A +0.000,E1 +46.501,E3 +56802.798,E4 +0.000} C_DIS
LIN {X -190.147,Y +401.077,Z +0.000,A +0.000,E1 +46.499,E3 +56817.839,E4 +0.000} C_DIS
LIN {X -190.159,Y +390.929,Z +0.000,A +0.000,E1 +46.494,E3 +56830.805,E4 +0.000} C_DIS
LIN {X -190.174,Y +383.973,Z +0.000,A +0.000,E1 +46.484,E3 +56839.698,E4 +0.000} C_DIS
LIN {X -190.200,Y +373.815,Z +0.000,A +0.000,E1 +46.448,E3 +56852.703,E4 +0.000} C_DIS
LIN {X -190.154,Y +361.003,Z +0.000,A +0.000,E1 +46.303,E3 +56869.197,E4 +0.000} C_DIS
LIN {X -189.772,Y +350.660,Z +0.000,A +0.049,E1 +45.996,E3 +56882.736,E4 +0.000} C_DIS
LIN {X -189.325,Y +346.917,Z +0.000,A +0.243,E1 +45.771,E3 +56887.805,E4 +0.000} C_DIS
LIN {X -188.196,Y +342.754,Z +0.000,A +1.966,E1 +45.249,E3 +56893.813,E4 +0.000} C_DIS
LIN {X -185.199,Y +337.023,Z +0.000,A +6.630,E1 +43.793,E3 +56903.187,E4 +0.000} C_DIS
LIN {X -181.141,Y +331.596,Z +0.000,A +12.274,E1 +41.569,E3 +56913.747,E4 +0.000} C_DIS
LIN {X -176.762,Y +326.804,Z +0.000,A +17.560,E1 +38.898,E3 +56925.171,E4 +0.000} C_DIS
LIN {X -172.184,Y +322.578,Z +0.000,A +19.859,E1 +36.197,E3 +56937.901,E4 +0.000} C_DIS
LIN {X -165.998,Y +317.874,Z +0.000,A +20.000,E1 +32.027,E3 +56957.659,E4 +0.000} C_DIS
LIN {X -160.137,Y +314.334,Z +0.000,A +20.000,E1 +26.368,E3 +56982.028,E4 +0.000} C_DIS
LIN {X -155.624,Y +312.245,Z +0.000,A +20.000,E1 +19.506,E3 +57010.704,E4 +0.000} C_DIS
LIN {X -153.557,Y +311.879,Z +0.000,A +20.000,E1 +11.113,E3 +57046.459,E4 +0.000} C_DIS
LIN {X -155.320,Y +313.348,Z +0.000,A +20.000,E1 +3.401,E3 +57079.643,E4 +0.000} C_DIS
LIN {X -160.005,Y +315.804,Z +0.000,A +20.000,E1 -4.720,E3 +57110.021,E4 +0.000} C_DIS
LIN {X -164.504,Y +318.255,Z +0.000,A +20.000,E1 -10.663,E3 +57129.390,E4 +0.000} C_DIS
LIN {X -170.340,Y +322.684,Z +0.000,A +20.000,E1 -17.457,E3 +57149.422,E4 +0.000} C_DIS
LIN {X -175.568,Y +329.106,Z +0.000,A +20.000,E1 -24.747,E3 +57166.656,E4 +0.000} C_DIS
LIN {X -184.074,Y +340.065,Z +0.000,A +20.000,E1 -33.664,E3 +57189.596,E4 +0.000} C_DIS
LIN {X -190.779,Y +351.388,Z +0.000,A +20.000,E1 -40.083,E3 +57207.374,E4 +0.000} C_DIS
LIN {X -195.254,Y +362.955,Z +0.000,A +20.000,E1 -44.515,E3 +57222.127,E4 +0.000} C_DIS
LIN {X -197.754,Y +374.780,Z +0.000,A +20.000,E1 -47.450,E3 +57235.549,E4 +0.000} C_DIS
LIN {X -198.310,Y +383.215,Z +0.000,A +19.956,E1 -48.698,E3 +57244.673,E4 +0.000} C_DIS
LIN {X -197.912,Y +391.275,Z +0.000,A +18.601,E1 -49.158,E3 +57253.391,E4 +0.000} C_DIS
LIN {X -196.679,Y +398.944,Z +0.000,A +13.989,E1 -48.784,E3 +57261.945,E4 +0.000} C_DIS
LIN {X -194.742,Y +406.288,Z +0.000,A +8.476,E1 -48.001,E3 +57270.628,E4 +0.000} C_DIS
LIN {X -192.748,Y +413.472,Z +0.000,A +3.905,E1 -47.267,E3 +57279.638,E4 +0.000} C_DIS
LIN {X -191.781,Y +419.162,Z +0.000,A +1.739,E1 -46.975,E3 +57286.906,E4 +0.000} C_DIS
LIN {X -190.795,Y +430.646,Z +0.000,A +0.152,E1 -46.707,E3 +57301.567,E4 +0.000} C_DIS
LIN {X -190.395,Y +441.145,Z +0.000,A +0.001,E1 -46.583,E3 +57314.960,E4 +0.000} C_DIS
LIN {X -190.239,Y +451.150,Z +0.000,A -0.000,E1 -46.528,E3 +57327.728,E4 +0.000} C_DIS
LIN {X -190.161,Y +465.026,Z +0.000,A -0.000,E1 -46.506,E3 +57345.443,E4 +0.000} C_DIS
LIN {X -190.142,Y +1057.148,Z +0.000,A -0.000,E1 -46.500,E3 +58101.649,E4 +0.000} C_DIS
LIN {X -190.147,Y +1068.924,Z +0.000,A -0.000,E1 -46.499,E3 +58116.690,E4 +0.000} C_DIS
LIN {X -190.159,Y +1079.072,Z +0.000,A -0.000,E1 -46.493,E3 +58129.655,E4 +0.000} C_DIS
LIN {X -190.174,Y +1086.028,Z +0.000,A -0.000,E1 -46.483,E3 +58138.549,E4 +0.000} C_DIS
LIN {X -190.200,Y +1096.186,Z +0.000,A -0.000,E1 -46.448,E3 +58151.553,E4 +0.000} C_DIS
LIN {X -190.154,Y +1108.998,Z +0.000,A -0.054,E1 -46.295,E3 +58168.048,E4 +0.000} C_DIS
LIN {X -189.772,Y +1119.341,Z +0.000,A -0.752,E1 -45.902,E3 +58181.586,E4 +0.000} C_DIS
LIN {X -189.097,Y +1124.276,Z +0.000,A -2.508,E1 -45.397,E3 +58188.318,E4 +0.000} C_DIS
LIN {X -187.410,Y +1129.069,Z +0.000,A -5.304,E1 -44.585,E3 +58195.491,E4 +0.000} C_DIS
LIN {X -183.899,Y +1134.873,Z +0.000,A -10.372,E1 -42.805,E3 +58205.497,E4 +0.000} C_DIS
LIN {X -179.711,Y +1140.065,Z +0.000,A -15.940,E1 -40.393,E3 +58216.283,E4 +0.000} C_DIS
LIN {X -176.763,Y +1143.197,Z +0.000,A -18.748,E1 -38.674,E3 +58224.021,E4 +0.000} C_DIS
LIN {X -172.185,Y +1147.423,Z +0.000,A -19.971,E1 -36.175,E3 +58236.751,E4 +0.000} C_DIS
LIN {X -165.999,Y +1152.127,Z +0.000,A -20.000,E1 -32.027,E3 +58256.509,E4 +0.000} C_DIS
LIN {X -160.138,Y +1155.667,Z +0.000,A -20.000,E1 -26.368,E3 +58280.879,E4 +0.000} C_DIS
LIN {X -155.625,Y +1157.756,Z +0.000,A -20.000,E1 -19.505,E3 +58309.555,E4 +0.000} C_DIS
LIN {X -153.552,Y +1158.113,Z +0.000,A -20.000,E1 -11.113,E3 +58345.306,E4 +0.000} C_DIS
LIN {X -156.311,Y +1155.540,Z +0.000,A -20.000,E1 -0.839,E3 +58388.666,E4 +0.000} C_DIS
LIN {X -161.281,Y +1151.851,Z +0.000,A -20.000,E1 +7.737,E3 +58418.565,E4 +0.000} C_DIS
LIN {X -167.493,Y +1147.157,Z +0.000,A -20.000,E1 +16.195,E3 +58443.004,E4 +0.000} C_DIS
LIN {X -173.235,Y +1142.221,Z +0.000,A -20.000,E1 +22.930,E3 +58460.306,E4 +0.000} C_DIS
LIN {X -181.123,Y +1133.734,Z +0.000,A -20.000,E1 +30.868,E3 +58481.062,E4 +0.000} C_DIS
LIN {X -189.654,Y +1120.856,Z +0.000,A -20.000,E1 +39.018,E3 +58503.076,E4 +0.000} C_DIS
LIN {X -195.246,Y +1107.046,Z +0.000,A -20.000,E1 +44.515,E3 +58520.978,E4 +0.000} C_DIS
LIN {X -198.051,Y +1092.368,Z +0.000,A -20.000,E1 +47.947,E3 +58537.504,E4 +0.000} C_DIS
LIN {X -198.143,Y +1081.370,Z +0.000,A -19.806,E1 +49.153,E3 +58549.365,E4 +0.000} C_DIS
LIN {X -197.177,Y +1073.569,Z +0.000,A -17.356,E1 +49.162,E3 +58557.949,E4 +0.000} C_DIS
LIN {X -195.448,Y +1066.139,Z +0.000,A -12.154,E1 +48.512,E3 +58566.544,E4 +0.000} C_DIS
LIN {X -193.346,Y +1058.941,Z +0.000,A -7.133,E1 +47.724,E3 +58575.424,E4 +0.000} C_DIS
LIN {X -191.781,Y +1050.839,Z +0.000,A -3.715,E1 +47.274,E3 +58585.757,E4 +0.000} C_DIS
LIN {X -190.795,Y +1039.355,Z +0.000,A -0.983,E1 +46.842,E3 +58600.417,E4 +0.000} C_DIS
LIN {X -190.395,Y +1028.856,Z +0.000,A -0.089,E1 +46.598,E3 +58613.811,E4 +0.000} C_DIS
LIN {X -190.239,Y +1018.851,Z +0.000,A -0.004,E1 +46.529,E3 +58626.579,E4 +0.000} C_DIS
LIN {X -190.161,Y +1004.975,Z +0.000,A +0.000,E1 +46.506,E3 +58644.293,E4 +0.000} C_DIS
LIN {X -190.142,Y +412.853,Z +0.000,A +0.000,E1 +46.501,E3 +59400.499,E4 +0.000} C_DIS
LIN {X -190.147,Y +401.077,Z +0.000,A +0.000,E1 +46.499,E3 +59415.540,E4 +0.000} C_DIS
LIN {X -190.159,Y +390.929,Z +0.000,A +0.000,E1 +46.494,E3 +59428.506,E4 +0.000} C_DIS
LIN {X -190.174,Y +383.973,Z +0.000,A +0.000,E1 +46.484,E3 +59437.399,E4 +0.000} C_DIS
LIN {X -190.200,Y +373.815,Z +0.000,A +0.000,E1 +46.448,E3 +59450.404,E4 +0.000} C_DIS
LIN {X -190.154,Y +361.003,Z +0.000,A +0.000,E1 +46.303,E3 +59466.898,E4 +0.000} C_DIS
LIN {X -189.772,Y +350.660,Z +0.000,A +0.049,E1 +45.996,E3 +59480.437,E4 +0.000} C_DIS
LIN {X -189.325,Y +346.917,Z +0.000,A +0.243,E1 +45.771,E3 +59485.506,E4 +0.000} C_DIS
LIN {X -188.196,Y +342.754,Z +0.000,A +1.966,E1 +45.249,E3 +59491.514,E4 +0.000} C_DIS
LIN {X -185.199,Y +337.023,Z +0.000,A +6.630,E1 +43.793,E3 +59500.888,E4 +0.000} C_DIS
LIN {X -181.141,Y +331.596,Z +0.000,A +12.274,E1 +41.569,E3 +59511.448,E4 +0.000} C_DIS
LIN {X -176.762,Y +326.804,Z +0.000,A +17.560,E1 +38.898,E3 +59522.872,E4 +0.000} C_DIS
LIN {X -172.184,Y +322.578,Z +0.000,A +19.859,E1 +36.197,E3 +59535.602,E4 +0.000} C_DIS
LIN {X -165.998,Y +317.874,Z +0.000,A +20.000,E1 +32.027,E3 +59555.360,E4 +0.000} C_DIS
LIN {X -160.137,Y +314.334,Z +0.000,A +20.000,E1 +26.368,E3 +59579.729,E4 +0.000} C_DIS
LIN {X -155.624,Y +312.245,Z +0.000,A +20.000,E1 +19.506,E3 +59608.405,E4 +0.000} C_DIS
LIN {X -153.557,Y +311.879,Z +0.000,A +20.000,E1 +11.113,E3 +59644.160,E4 +0.000} C_DIS
LIN {X -155.320,Y +313.348,Z +0.000,A +20.000,E1 +3.401,E3 +59677.344,E4 +0.000} C_DIS
LIN {X -160.005,Y +315.804,Z +0.000,A +20.000,E1 -4.720,E3 +59707.722,E4 +0.000} C_DIS
LIN {X -164.504,Y +318.255,Z +0.000,A +20.000,E1 -10.663,E3 +59727.091,E4 +0.000} C_DIS
LIN {X -170.340,Y +322.684,Z +0.000,A +20.000,E1 -17.457,E3 +59747.123,E4 +0.000} C_DIS
LIN {X -175.568,Y +329.106,Z +0.000,A +20.000,E1 -24.747,E3 +59764.357,E4 +0.000} C_DIS
LIN {X -184.074,Y +340.065,Z +0.000,A +20.000,E1 -33.664,E3 +59787.297,E4 +0.000} C_DIS
LIN {X -190.779,Y +351.388,Z +0.000,A +20.000,E1 -40.083,E3 +59805.075,E4 +0.000} C_DIS
LIN {X -195.254,Y +362.955,Z +0.000,A +20.000,E1 -44.515,E3 +59819.828,E4 +0.000} C_DIS
LIN {X -197.754,Y +374.780,Z +0.000,A +20.000,E1 -47.450,E3 +59833.250,E4 +0.000} C_DIS
LIN {X -198.310,Y +383.215,Z +0.000,A +19.956,E1 -48.698,E3 +59842.374,E4 +0.000} C_DIS
LIN {X -197.912,Y +391.275,Z +0.000,A +18.601,E1 -49.158,E3 +59851.092,E4 +0.000} C_DIS
LIN {X -196.679,Y +398.944,Z +0.000,A +13.989,E1 -48.784,E3 +59859.646,E4 +0.000} C_DIS
LIN {X -194.742,Y +406.288,Z +0.000,A +8.476,E1 -48.001,E3 +59868.329,E4 +0.000} C_DIS
LIN {X -192.748,Y +413.472,Z +0.000,A +3.905,E1 -47.267,E3 +59877.339,E4 +0.000} C_DIS
LIN {X -191.781,Y +419.162,Z +0.000,A +1.739,E1 -46.975,E3 +59884.607,E4 +0.000} C_DIS
LIN {X -190.795,Y +430.646,Z +0.000,A +0.152,E1 -46.707,E3 +59899.268,E4 +0.000} C_DIS
LIN {X -190.395,Y +441.145,Z +0.000,A +0.001,E1 -46.583,E3 +59912.661,E4 +0.000} C_DIS
LIN {X -190.239,Y +451.150,Z +0.000,A -0.000,E1 -46.528,E3 +59925.429,E4 +0.000} C_DIS
LIN {X -190.161,Y +465.026,Z +0.000,A -0.000,E1 -46.506,E3 +59943.144,E4 +0.000} C_DIS
LIN {X -190.142,Y +1057.148,Z +0.000,A -0.000,E1 -46.500,E3 +60699.350,E4 +0.000} C_DIS
LIN {X -190.147,Y +1068.924,Z +0.000,A -0.000,E1 -46.499,E3 +60714.391,E4 +0.000} C_DIS
LIN {X -190.159,Y +1079.072,Z +0.000,A -0.000,E1 -46.493,E3 +60727.356,E4 +0.000} C_DIS
LIN {X -190.174,Y +1086.028,Z +0.000,A -0.000,E1 -46.483,E3 +60736.250,E4 +0.000} C_DIS
LIN {X -190.200,Y +1096.186,Z +0.000,A -0.000,E1 -46.448,E3 +60749.254,E4 +0.000} C_DIS
LIN {X -190.154,Y +1108.998,Z +0.000,A -0.054,E1 -46.295,E3 +60765.749,E4 +0.000} C_DIS
LIN {X -189.772,Y +1119.341,Z +0.000,A -0.752,E1 -45.902,E3 +60779.287,E4 +0.000} C_DIS
LIN {X -189.097,Y +1124.276,Z +0.000,A -2.508,E1 -45.397,E3 +60786.019,E4 +0.000} C_DIS
LIN {X -187.410,Y +1129.069,Z +0.000,A -5.304,E1 -44.585,E3 +60793.192,E4 +0.000} C_DIS
LIN {X -183.899,Y +1134.873,Z +0.000,A -10.372,E1 -42.805,E3 +60803.198,E4 +0.000} C_DIS
LIN {X -179.711,Y +1140.065,Z +0.000,A -15.940,E1 -40.393,E3 +60813.984,E4 +0.000} C_DIS
LIN {X -176.763,Y +1143.197,Z +0.000,A -18.748,E1 -38.674,E3 +60821.722,E4 +0.000} C_DIS
LIN {X -172.185,Y +1147.423,Z +0.000,A -19.971,E1 -36.175,E3 +60834.452,E4 +0.000} C_DIS
LIN {X -165.999,Y +1152.127,Z +0.000,A -20.000,E1 -32.027,E3 +60854.210,E4 +0.000} C_DIS
LIN {X -160.138,Y +1155.667,Z +0.000,A -20.000,E1 -26.368,E3 +60878.580,E4 +0.000} C_DIS
LIN {X -155.625,Y +1157.756,Z +0.000,A -20.000,E1 -19.505,E3 +60907.256,E4 +0.000} C_DIS
LIN {X -153.552,Y +1158.113,Z +0.000,A -20.000,E1 -11.113,E3 +60943.007,E4 +0.000} C_DIS
LIN {X -156.311,Y +1155.540,Z +0.000,A -20.000,E1 -0.839,E3 +60986.367,E4 +0.000} C_DIS
LIN {X -161.281,Y +1151.851,Z +0.000,A -20.000,E1 +7.737,E3 +61016.266,E4 +0.000} C_DIS
LIN {X -167.493,Y +1147.157,Z +0.000,A -20.000,E1 +16.195,E3 +61040.705,E4 +0.000} C_DIS
LIN {X -173.235,Y +1142.221,Z +0.000,A -20.000,E1 +22.930,E3 +61058.007,E4 +0.000} C_DIS
LIN {X -181.123,Y +1133.734,Z +0.000,A -20.000,E1 +30.868,E3 +61078.763,E4 +0.000} C_DIS
LIN {X -189.654,Y +1120.856,Z +0.000,A -20.000,E1 +39.018,E3 +61100.777,E4 +0.000} C_DIS
LIN {X -195.246,Y +1107.046,Z +0.000,A -20.000,E1 +44.515,E3 +61118.679,E4 +0.000} C_DIS
LIN {X -198.051,Y +1092.368,Z +0.000,A -20.000,E1 +47.947,E3 +61135.205,E4 +0.000} C_DIS
LIN {X -198.143,Y +1081.370,Z +0.000,A -19.806,E1 +49.153,E3 +61147.066,E4 +0.000} C_DIS
LIN {X -197.177,Y +1073.569,Z +0.000,A -17.356,E1 +49.162,E3 +61155.650,E4 +0.000} C_DIS
LIN {X -195.448,Y +1066.139,Z +0.000,A -12.154,E1 +48.512,E3 +61164.245,E4 +0.000} C_DIS
LIN {X -193.346,Y +1058.941,Z +0.000,A -7.133,E1 +47.724,E3 +61173.125,E4 +0.000} C_DIS
LIN {X -191.781,Y +1050.839,Z +0.000,A -3.715,E1 +47.274,E3 +61183.458,E4 +0.000} C_DIS
LIN {X -190.795,Y +1039.355,Z +0.000,A -0.983,E1 +46.842,E3 +61198.118,E4 +0.000} C_DIS
LIN {X -190.395,Y +1028.856,Z +0.000,A -0.089,E1 +46.598,E3 +61211.512,E4 +0.000} C_DIS
LIN {X -190.239,Y +1018.851,Z +0.000,A -0.004,E1 +46.529,E3 +61224.280,E4 +0.000} C_DIS
LIN {X -190.161,Y +1004.975,Z +0.000,A +0.000,E1 +46.506,E3 +61241.994,E4 +0.000} C_DIS
LIN {X -190.142,Y +412.853,Z +0.000,A +0.000,E1 +46.501,E3 +61998.200,E4 +0.000} C_DIS
LIN {X -190.147,Y +401.077,Z +0.000,A +0.000,E1 +46.499,E3 +62013.241,E4 +0.000} C_DIS
LIN {X -190.159,Y +390.929,Z +0.000,A +0.000,E1 +46.494,E3 +62026.207,E4 +0.000} C_DIS
LIN {X -190.174,Y +383.973,Z +0.000,A +0.000,E1 +46.484,E3 +62035.100,E4 +0.000} C_DIS
LIN {X -190.200,Y +373.815,Z +0.000,A +0.000,E1 +46.448,E3 +62048.105,E4 +0.000} C_DIS
LIN {X -190.154,Y +361.003,Z +0.000,A +0.000,E1 +46.303,E3 +62064.599,E4 +0.000} C_DIS
LIN {X -189.772,Y +350.660,Z +0.000,A +0.049,E1 +45.996,E3 +62078.138,E4 +0.000} C_DIS
LIN {X -189.325,Y +346.917,Z +0.000,A +0.243,E1 +45.771,E3 +62083.207,E4 +0.000} C_DIS
LIN {X -188.196,Y +342.754,Z +0.000,A +1.966,E1 +45.249,E3 +62089.215,E4 +0.000} C_DIS
LIN {X -185.199,Y +337.023,Z +0.000,A +6.630,E1 +43.793,E3 +62098.589,E4 +0.000} C_DIS
LIN {X -181.141,Y +331.596,Z +0.000,A +12.274,E1 +41.569,E3 +62109.149,E4 +0.000} C_DIS
LIN {X -176.762,Y +326.804,Z +0.000,A +17.560,E1 +38.898,E3 +62120.573,E4 +0.000} C_DIS
LIN {X -172.184,Y +322.578,Z +0.000,A +19.859,E1 +36.197,E3 +62133.303,E4 +0.000} C_DIS
LIN {X -165.998,Y +317.874,Z +0.000,A +20.000,E1 +32.027,E3 +62153.061,E4 +0.000} C_DIS
LIN {X -160.137,Y +314.334,Z +0.000,A +20.000,E1 +26.368,E3 +62177.430,E4 +0.000} C_DIS
LIN {X -155.624,Y +312.245,Z +0.000,A +20.000,E1 +19.506,E3 +62206.106,E4 +0.000} C_DIS
LIN {X -153.557,Y +311.879,Z +0.000,A +20.000,E1 +11.113,E3 +62241.861,E4 +0.000} C_DIS
LIN {X -155.320,Y +313.348,Z +0.000,A +20.000,E1 +3.401,E3 +62275.045,E4 +0.000} C_DIS
LIN {X -160.005,Y +315.804,Z +0.000,A +20.000,E1 -4.720,E3 +62305.423,E4 +0.000} C_DIS
LIN {X -164.504,Y +318.255,Z +0.000,A +20.000,E1 -10.663,E3 +62324.792,E4 +0.000} C_DIS
LIN {X -170.340,Y +322.684,Z +0.000,A +20.000,E1 -17.457,E3 +62344.824,E4 +0.000} C_DIS
LIN {X -175.568,Y +329.106,Z +0.000,A +20.000,E1 -24.747,E3 +62362.058,E4 +0.000} C_DIS
LIN {X -184.074,Y +340.065,Z +0.000,A +20.000,E1 -33.664,E3 +62384.998,E4 +0.000} C_DIS
LIN {X -190.779,Y +351.388,Z +0.000,A +20.000,E1 -40.083,E3 +62402.776,E4 +0.000} C_DIS
LIN {X -195.254,Y +362.955,Z +0.000,A +20.000,E1 -44.515,E3 +62417.529,E4 +0.000} C_DIS
LIN {X -197.754,Y +374.780,Z +0.000,A +20.000,E1 -47.450,E3 +62430.951,E4 +0.000} C_DIS
LIN {X -198.310,Y +383.215,Z +0.000,A +19.956,E1 -48.698,E3 +62440.075,E4 +0.000} C_DIS
LIN {X -197.912,Y +391.275,Z +0.000,A +18.601,E1 -49.158,E3 +62448.793,E4 +0.000} C_DIS
LIN {X -196.679,Y +398.944,Z +0.000,A +13.989,E1 -48.784,E3 +62457.347,E4 +0.000} C_DIS
LIN {X -194.742,Y +406.288,Z +0.000,A +8.476,E1 -48.001,E3 +62466.030,E4 +0.000} C_DIS
LIN {X -192.748,Y +413.472,Z +0.000,A +3.905,E1 -47.267,E3 +62475.040,E4 +0.000} C_DIS
LIN {X -191.781,Y +419.162,Z +0.000,A +1.739,E1 -46.975,E3 +62482.308,E4 +0.000} C_DIS
LIN {X -190.795,Y +430.646,Z +0.000,A +0.152,E1 -46.707,E3 +62496.969,E4 +0.000} C_DIS
LIN {X -190.395,Y +441.145,Z +0.000,A +0.001,E1 -46.583,E3 +62510.362,E4 +0.000} C_DIS
LIN {X -190.239,Y +451.150,Z +0.000,A -0.000,E1 -46.528,E3 +62523.130,E4 +0.000} C_DIS
LIN {X -190.161,Y +465.026,Z +0.000,A -0.000,E1 -46.506,E3 +62540.845,E4 +0.000} C_DIS
LIN {X -190.142,Y +1057.148,Z +0.000,A -0.000,E1 -46.500,E3 +63297.051,E4 +0.000} C_DIS
LIN {X -190.147,Y +1068.924,Z +0.000,A -0.000,E1 -46.499,E3 +63312.092,E4 +0.000} C_DIS
LIN {X -190.159,Y +1079.072,Z +0.000,A -0.000,E1 -46.493,E3 +63325.057,E4 +0.000} C_DIS
LIN {X -190.174,Y +1086.028,Z +0.000,A -0.000,E1 -46.483,E3 +63333.951,E4 +0.000} C_DIS
LIN {X -190.200,Y +1096.186,Z +0.000,A -0.000,E1 -46.448,E3 +63346.955,E4 +0.000} C_DIS
LIN {X -190.154,Y +1108.998,Z +0.000,A -0.054,E1 -46.295,E3 +63363.450,E4 +0.000} C_DIS
LIN {X -189.772,Y +1119.341,Z +0.000,A -0.752,E1 -45.902,E3 +63376.988,E4 +0.000} C_DIS
LIN {X -189.097,Y +1124.276,Z +0.000,A -2.508,E1 -45.397,E3 +63383.720,E4 +0.000} C_DIS
LIN {X -187.410,Y +1129.069,Z +0.000,A -5.304,E1 -44.585,E3 +63390.893,E4 +0.000} C_DIS
LIN {X -183.899,Y +1134.873,Z +0.000,A -10.372,E1 -42.805,E3 +63400.899,E4 +0.000} C_DIS
LIN {X -179.711,Y +1140.065,Z +0.000,A -15.940,E1 -40.393,E3 +63411.685,E4 +0.000} C_DIS
LIN {X -176.763,Y +1143.197,Z +0.000,A -18.748,E1 -38.674,E3 +63419.423,E4 +0.000} C_DIS
LIN {X -172.185,Y +1147.423,Z +0.000,A -19.971,E1 -36.175,E3 +63432.153,E4 +0.000} C_DIS
LIN {X -165.999,Y +1152.127,Z +0.000,A -20.000,E1 -32.027,E3 +63451.911,E4 +0.000} C_DIS
LIN {X -160.138,Y +1155.667,Z +0.000,A -20.000,E1 -26.368,E3 +63476.281,E4 +0.000} C_DIS
LIN {X -155.625,Y +1157.756,Z +0.000,A -20.000,E1 -19.505,E3 +63504.957,E4 +0.000} C_DIS
LIN {X -153.552,Y +1158.113,Z +0.000,A -20.000,E1 -11.113,E3 +63540.708,E4 +0.000} C_DIS
LIN {X -156.311,Y +1155.540,Z +0.000,A -20.000,E1 -0.839,E3 +63584.068,E4 +0.000} C_DIS
LIN {X -161.281,Y +1151.851,Z +0.000,A -20.000,E1 +7.737,E3 +63613.967,E4 +0.000} C_DIS
LIN {X -167.493,Y +1147.157,Z +0.000,A -20.000,E1 +16.195,E3 +63638.406,E4 +0.000} C_DIS
LIN {X -173.235,Y +1142.221,Z +0.000,A -20.000,E1 +22.930,E3 +63655.708,E4 +0.000} C_DIS
LIN {X -181.123,Y +1133.734,Z +0.000,A -20.000,E1 +30.868,E3 +63676.464,E4 +0.000} C_DIS
LIN {X -189.654,Y +1120.856,Z +0.000,A -20.000,E1 +39.018,E3 +63698.478,E4 +0.000} C_DIS
LIN {X -195.246,Y +1107.046,Z +0.000,A -20.000,E1 +44.515,E3 +63716.380,E4 +0.000} C_DIS
LIN {X -198.051,Y +1092.368,Z +0.000,A -20.000,E1 +47.947,E3 +63732.906,E4 +0.000} C_DIS
LIN {X -198.143,Y +1081.370,Z +0.000,A -19.806,E1 +49.153,E3 +63744.767,E4 +0.000} C_DIS
LIN {X -197.177,Y +1073.569,Z +0.000,A -17.356,E1 +49.162,E3 +63753.351,E4 +0.000} C_DIS
LIN {X -195.448,Y +1066.139,Z +0.000,A -12.154,E1 +48.512,E3 +63761.946,E4 +0.000} C_DIS
LIN {X -193.346,Y +1058.941,Z +0.000,A -7.133,E1 +47.724,E3 +63770.826,E4 +0.000} C_DIS
LIN {X -191.781,Y +1050.839,Z +0.000,A -3.715,E1 +47.274,E3 +63781.159,E4 +0.000} C_DIS
LIN {X -190.795,Y +1039.355,Z +0.000,A -0.983,E1 +46.842,E3 +63795.819,E4 +0.000} C_DIS
LIN {X -190.395,Y +1028.856,Z +0.000,A -0.089,E1 +46.598,E3 +63809.213,E4 +0.000} C_DIS
LIN {X -190.239,Y +1018.851,Z +0.000,A -0.004,E1 +46.529,E3 +63821.981,E4 +0.000} C_DIS
LIN {X -190.161,Y +1004.975,Z +0.000,A +0.000,E1 +46.506,E3 +63839.695,E4 +0.000} C_DIS
LIN {X -190.142,Y +412.853,Z +0.000,A +0.000,E1 +46.501,E3 +64595.901,E4 +0.000} C_DIS
LIN {X -190.147,Y +401.077,Z +0.000,A +0.000,E1 +46.499,E3 +64610.942,E4 +0.000} C_DIS
LIN {X -190.159,Y +390.929,Z +0.000,A +0.000,E1 +46.494,E3 +64623.908,E4 +0.000} C_DIS
LIN {X -190.174,Y +383.973,Z +0.000,A +0.000,E1 +46.484,E3 +64632.801,E4 +0.000} C_DIS
LIN {X -190.200,Y +373.815,Z +0.000,A +0.000,E1 +46.448,E3 +64645.806,E4 +0.000} C_DIS
LIN {X -190.154,Y +361.003,Z +0.000,A +0.000,E1 +46.303,E3 +64662.300,E4 +0.000} C_DIS
LIN {X -189.772,Y +350.660,Z +0.000,A +0.049,E1 +45.996,E3 +64675.839,E4 +0.000} C_DIS
LIN {X -189.325,Y +346.917,Z +0.000,A +0.243,E1 +45.771,E3 +64680.908,E4 +0.000} C_DIS
LIN {X -188.196,Y +342.754,Z +0.000,A +1.966,E1 +45.249,E3 +64686.916,E4 +0.000} C_DIS
LIN {X -185.199,Y +337.023,Z +0.000,A +6.630,E1 +43.793,E3 +64696.290,E4 +0.000} C_DIS
LIN {X -181.141,Y +331.596,Z +0.000,A +12.274,E1 +41.569,E3 +64706.850,E4 +0.000} C_DIS
LIN {X -176.762,Y +326.804,Z +0.000,A +17.560,E1 +38.898,E3 +64718.274,E4 +0.000} C_DIS
LIN {X -172.184,Y +322.578,Z +0.000,A +19.859,E1 +36.197,E3 +64731.004,E4 +0.000} C_DIS
LIN {X -165.998,Y +317.874,Z +0.000,A +20.000,E1 +32.027,E3 +64750.762,E4 +0.000} C_DIS
LIN {X -160.137,Y +314.334,Z +0.000,A +20.000,E1 +26.368,E3 +64775.131,E4 +0.000} C_DIS
LIN {X -155.624,Y +312.245,Z +0.000,A +20.000,E1 +19.506,E3 +64803.807,E4 +0.000} C_DIS
LIN {X -153.557,Y +311.879,Z +0.000,A +20.000,E1 +11.113,E3 +64839.562,E4 +0.000} C_DIS
LIN {X -155.320,Y +313.348,Z +0.000,A +20.000,E1 +3.401,E3 +64872.746,E4 +0.000} C_DIS
LIN {X -160.005,Y +315.804,Z +0.000,A +20.000,E1 -4.720,E3 +64903.124,E4 +0.000} C_DIS
LIN {X -164.504,Y +318.255,Z +0.000,A +20.000,E1 -10.663,E3 +64922.493,E4 +0.000} C_DIS
LIN {X -170.340,Y +322.684,Z +0.000,A +20.000,E1 -17.457,E3 +64942.525,E4 +0.000} C_DIS
LIN {X -175.568,Y +329.106,Z +0.000,A +20.000,E1 -24.747,E3 +64959.759,E4 +0.000} C_DIS
LIN {X -184.074,Y +340.065,Z +0.000,A +20.000,E1 -33.664,E3 +64982.699,E4 +0.000} C_DIS
LIN {X -190.779,Y +351.388,Z +0.000,A +20.000,E1 -40.083,E3 +65000.477,E4 +0.000} C_DIS
LIN {X -195.254,Y +362.955,Z +0.000,A +20.000,E1 -44.515,E3 +65015.230,E4 +0.000} C_DIS
LIN {X -197.754,Y +374.780,Z +0.000,A +20.000,E1 -47.450,E3 +65028.652,E4 +0.000} C_DIS
LIN {X -198.310,Y +383.215,Z +0.000,A +19.956,E1 -48.698,E3 +65037.776,E4 +0.000} C_DIS
LIN {X -197.912,Y +391.275,Z +0.000,A +18.601,E1 -49.158,E3 +65046.494,E4 +0.000} C_DIS
LIN {X -196.679,Y +398.944,Z +0.000,A +13.989,E1 -48.784,E3 +65055.048,E4 +0.000} C_DIS
LIN {X -194.742,Y +406.288,Z +0.000,A +8.476,E1 -48.001,E3 +65063.731,E4 +0.000} C_DIS
LIN {X -192.748,Y +413.472,Z +0.000,A +3.905,E1 -47.267,E3 +65072.741,E4 +0.000} C_DIS
LIN {X -191.781,Y +419.162,Z +0.000,A +1.739,E1 -46.975,E3 +65080.009,E4 +0.000} C_DIS
LIN {X -190.795,Y +430.646,Z +0.000,A +0.152,E1 -46.707,E3 +65094.670,E4 +0.000} C_DIS
LIN {X -190.395,Y +441.145,Z +0.000,A +0.001,E1 -46.583,E3 +65108.063,E4 +0.000} C_DIS
LIN {X -190.239,Y +451.150,Z +0.000,A -0.000,E1 -46.528,E3 +65120.831,E4 +0.000} C_DIS
LIN {X -190.161,Y +465.026,Z +0.000,A -0.000,E1 -46.506,E3 +65138.546,E4 +0.000} C_DIS
LIN {X -190.142,Y +1057.148,Z +0.000,A -0.000,E1 -46.500,E3 +65894.752,E4 +0.000} C_DIS
LIN {X -190.147,Y +1068.924,Z +0.000,A -0.000,E1 -46.499,E3 +65909.793,E4 +0.000} C_DIS
LIN {X -190.159,Y +1079.072,Z +0.000,A -0.000,E1 -46.493,E3 +65922.758,E4 +0.000} C_DIS
LIN {X -190.174,Y +1086.028,Z +0.000,A -0.000,E1 -46.483,E3 +65931.652,E4 +0.000} C_DIS
LIN {X -190.200,Y +1096.186,Z +0.000,A -0.000,E1 -46.448,E3 +65944.656,E4 +0.000} C_DIS
LIN {X -190.154,Y +1108.998,Z +0.000,A -0.054,E1 -46.295,E3 +65961.151,E4 +0.000} C_DIS
LIN {X -189.772,Y +1119.341,Z +0.000,A -0.752,E1 -45.902,E3 +65974.689,E4 +0.000} C_DIS
LIN {X -189.097,Y +1124.276,Z +0.000,A -2.508,E1 -45.397,E3 +65981.421,E4 +0.000} C_DIS
LIN {X -187.410,Y +1129.069,Z +0.000,A -5.304,E1 -44.585,E3 +65988.594,E4 +0.000} C_DIS
LIN {X -183.899,Y +1134.873,Z +0.000,A -10.372,E1 -42.805,E3 +65998.600,E4 +0.000} C_DIS
LIN {X -179.711,Y +1140.065,Z +0.000,A -15.940,E1 -40.393,E3 +66009.386,E4 +0.000} C_DIS
LIN {X -176.763,Y +1143.197,Z +0.000,A -18.748,E1 -38.674,E3 +66017.124,E4 +0.000} C_DIS
LIN {X -172.185,Y +1147.423,Z +0.000,A -19.971,E1 -36.175,E3 +66029.854,E4 +0.000} C_DIS
LIN {X -165.999,Y +1152.127,Z +0.000,A -20.000,E1 -32.027,E3 +66049.612,E4 +0.000} C_DIS
LIN {X -160.138,Y +1155.667,Z +0.000,A -20.000,E1 -26.368,E3 +66073.982,E4 +0.000} C_DIS
LIN {X -155.625,Y +1157.756,Z +0.000,A -20.000,E1 -19.505,E3 +66102.658,E4 +0.000} C_DIS
LIN {X -153.552,Y +1158.113,Z +0.000,A -20.000,E1 -11.113,E3 +66138.409,E4 +0.000} C_DIS
LIN {X -156.311,Y +1155.540,Z +0.000,A -20.000,E1 -0.839,E3 +66181.769,E4 +0.000} C_DIS
LIN {X -161.281,Y +1151.851,Z +0.000,A -20.000,E1 +7.737,E3 +66211.668,E4 +0.000} C_DIS
LIN {X -167.493,Y +1147.157,Z +0.000,A -20.000,E1 +16.195,E3 +66236.107,E4 +0.000} C_DIS
LIN {X -173.235,Y +1142.221,Z +0.000,A -20.000,E1 +22.930,E3 +66253.409,E4 +0.000} C_DIS
LIN {X -181.123,Y +1133.734,Z +0.000,A -20.000,E1 +30.868,E3 +66274.165,E4 +0.000} C_DIS
LIN {X -189.654,Y +1120.856,Z +0.000,A -20.000,E1 +39.018,E3 +66296.179,E4 +0.000} C_DIS
LIN {X -195.246,Y +1107.046,Z +0.000,A -20.000,E1 +44.515,E3 +66314.081,E4 +0.000} C_DIS
LIN {X -198.051,Y +1092.368,Z +0.000,A -20.000,E1 +47.947,E3 +66330.607,E4 +0.000} C_DIS
LIN {X -198.143,Y +1081.370,Z +0.000,A -19.806,E1 +49.153,E3 +66342.468,E4 +0.000} C_DIS
LIN {X -197.177,Y +1073.569,Z +0.000,A -17.356,E1 +49.162,E3 +66351.052,E4 +0.000} C_DIS
LIN {X -195.448,Y +1066.139,Z +0.000,A -12.154,E1 +48.512,E3 +66359.647,E4 +0.000} C_DIS
LIN {X -193.346,Y +1058.941,Z +0.000,A -7.133,E1 +47.724,E3 +66368.527,E4 +0.000} C_DIS
LIN {X -191.781,Y +1050.839,Z +0.000,A -3.715,E1 +47.274,E3 +66378.860,E4 +0.000} C_DIS
LIN {X -190.795,Y +1039.355,Z +0.000,A -0.983,E1 +46.842,E3 +66393.520,E4 +0.000} C_DIS
LIN {X -190.395,Y +1028.856,Z +0.000,A -0.089,E1 +46.598,E3 +66406.914,E4 +0.000} C_DIS
LIN {X -190.239,Y +1018.851,Z +0.000,A -0.004,E1 +46.529,E3 +66419.682,E4 +0.000} C_DIS
LIN {X -190.161,Y +1004.975,Z +0.000,A +0.000,E1 +46.506,E3 +66437.396,E4 +0.000} C_DIS
LIN {X -190.142,Y +412.853,Z +0.000,A +0.000,E1 +46.501,E3 +67193.602,E4 +0.000} C_DIS
LIN {X -190.147,Y +401.077,Z +0.000,A +0.000,E1 +46.499,E3 +67208.643,E4 +0.000} C_DIS
LIN {X -190.159,Y +390.929,Z +0.000,A +0.000,E1 +46.494,E3 +67221.609,E4 +0.000} C_DIS
LIN {X -190.174,Y +383.973,Z +0.000,A +0.000,E1 +46.484,E3 +67230.502,E4 +0.000} C_DIS
LIN {X -190.200,Y +373.815,Z +0.000,A +0.000,E1 +46.448,E3 +67243.507,E4 +0.000} C_DIS
LIN {X -190.154,Y +361.003,Z +0.000,A +0.000,E1 +46.303,E3 +67260.001,E4 +0.000} C_DIS
LIN {X -189.772,Y +350.660,Z +0.000,A +0.049,E1 +45.996,E3 +67273.540,E4 +0.000} C_DIS
LIN {X -189.325,Y +346.917,Z +0.000,A +0.243,E1 +45.771,E3 +67278.609,E4 +0.000} C_DIS
LIN {X -188.196,Y +342.754,Z +0.000,A +1.966,E1 +45.249,E3 +67284.617,E4 +0.000} C_DIS
LIN {X -185.199,Y +337.023,Z +0.000,A +6.630,E1 +43.793,E3 +67293.991,E4 +0.000} C_DIS
LIN {X -181.141,Y +331.596,Z +0.000,A +12.274,E1 +41.569,E3 +67304.551,E4 +0.000} C_DIS
LIN {X -176.762,Y +326.804,Z +0.000,A +17.560,E1 +38.898,E3 +67315.975,E4 +0.000} C_DIS
LIN {X -172.184,Y +322.578,Z +0.000,A +19.859,E1 +36.197,E3 +67328.705,E4 +0.000} C_DIS
LIN {X -165.998,Y +317.874,Z +0.000,A +20.000,E1 +32.027,E3 +67348.463,E4 +0.000} C_DIS
LIN {X -160.137,Y +314.334,Z +0.000,A +20.000,E1 +26.368,E3 +67372.832,E4 +0.000} C_DIS
LIN {X -155.624,Y +312.245,Z +0.000,A +20.000,E1 +19.506,E3 +67401.508,E4 +0.000} C_DIS
LIN {X -153.557,Y +311.879,Z +0.000,A +20.000,E1 +11.113,E3 +67437.263,E4 +0.000} C_DIS
LIN {X -155.320,Y +313.348,Z +0.000,A +20.000,E1 +3.401,E3 +67470.447,E4 +0.000} C_DIS
LIN {X -160.005,Y +315.804,Z +0.000,A +20.000,E1 -4.720,E3 +67500.825,E4 +0.000} C_DIS
LIN {X -164.504,Y +318.255,Z +0.000,A +20.000,E1 -10.663,E3 +67520.194,E4 +0.000} C_DIS
LIN {X -170.340,Y +322.684,Z +0.000,A +20.000,E1 -17.457,E3 +67540.226,E4 +0.000} C_DIS
LIN {X -175.568,Y +329.106,Z +0.000,A +20.000,E1 -24.747,E3 +67557.460,E4 +0.000} C_DIS
LIN {X -184.074,Y +340.065,Z +0.000,A +20.000,E1 -33.664,E3 +67580.400,E4 +0.000} C_DIS
LIN {X -190.779,Y +351.388,Z +0.000,A +20.000,E1 -40.083,E3 +67598.178,E4 +0.000} C_DIS
LIN {X -195.254,Y +362.955,Z +0.000,A +20.000,E1 -44.515,E3 +67612.931,E4 +0.000} C_DIS
LIN {X -197.754,Y +374.780,Z +0.000,A +20.000,E1 -47.450,E3 +67626.353,E4 +0.000} C_DIS
LIN {X -198.310,Y +383.215,Z +0.000,A +19.956,E1 -48.698,E3 +67635.477,E4 +0.000} C_DIS
LIN {X -197.912,Y +391.275,Z +0.000,A +18.601,E1 -49.158,E3 +67644.195,E4 +0.000} C_DIS
LIN {X -196.679,Y +398.944,Z +0.000,A +13.989,E1 -48.784,E3 +67652.749,E4 +0.000} C_DIS
LIN {X -194.742,Y +406.288,Z +0.000,A +8.476,E1 -48.001,E3 +67661.432,E4 +0.000} C_DIS
LIN {X -192.748,Y +413.472,Z +0.000,A +3.905,E1 -47.267,E3 +67670.442,E4 +0.000} C_DIS
LIN {X -191.781,Y +419.162,Z +0.000,A +1.739,E1 -46.975,E3 +67677.710,E4 +0.000} C_DIS
LIN {X -190.795,Y +430.646,Z +0.000,A +0.152,E1 -46.707,E3 +67692.371,E4 +0.000} C_DIS
LIN {X -190.395,Y +441.145,Z +0.000,A +0.001,E1 -46.583,E3 +67705.764,E4 +0.000} C_DIS
LIN {X -190.239,Y +451.150,Z +0.000,A -0.000,E1 -46.528,E3 +67718.532,E4 +0.000} C_DIS
LIN {X -190.161,Y +465.026,Z +0.000,A -0.000,E1 -46.506,E3 +67736.247,E4 +0.000} C_DIS
LIN {X -190.142,Y +1057.148,Z +0.000,A -0.000,E1 -46.500,E3 +68492.453,E4 +0.000} C_DIS
LIN {X -190.147,Y +1068.924,Z +0.000,A -0.000,E1 -46.499,E3 +68507.494,E4 +0.000} C_DIS
LIN {X -190.159,Y +1079.072,Z +0.000,A -0.000,E1 -46.493,E3 +68520.459,E4 +0.000} C_DIS
LIN {X -190.174,Y +1086.028,Z +0.000,A -0.000,E1 -46.483,E3 +68529.353,E4 +0.000} C_DIS
LIN {X -190.200,Y +1096.186,Z +0.000,A -0.000,E1 -46.448,E3 +68542.357,E4 +0.000} C_DIS
LIN {X -190.154,Y +1108.998,Z +0.000,A -0.054,E1 -46.295,E3 +68558.852,E4 +0.000} C_DIS
LIN {X -189.772,Y +1119.341,Z +0.000,A -0.752,E1 -45.902,E3 +68572.390,E4 +0.000} C_DIS
LIN {X -189.097,Y +1124.276,Z +0.000,A -2.508,E1 -45.397,E3 +68579.122,E4 +0.000} C_DIS
LIN {X -187.410,Y +1129.069,Z +0.000,A -5.304,E1 -44.585,E3 +68586.295,E4 +0.000} C_DIS
LIN {X -183.899,Y +1134.873,Z +0.000,A -10.372,E1 -42.805,E3 +68596.301,E4 +0.000} C_DIS
LIN {X -179.711,Y +1140.065,Z +0.000,A -15.940,E1 -40.393,E3 +68607.087,E4 +0.000} C_DIS
LIN {X -176.763,Y +1143.197,Z +0.000,A -18.748,E1 -38.674,E3 +68614.825,E4 +0.000} C_DIS
LIN {X -172.185,Y +1147.423,Z +0.000,A -19.971,E1 -36.175,E3 +68627.555,E4 +0.000} C_DIS
LIN {X -165.999,Y +1152.127,Z +0.000,A -20.000,E1 -32.027,E3 +68647.313,E4 +0.000} C_DIS
LIN {X -160.138,Y +1155.667,Z +0.000,A -20.000,E1 -26.368,E3 +68671.683,E4 +0.000} C_DIS
LIN {X -155.625,Y +1157.756,Z +0.000,A -20.000,E1 -19.505,E3 +68700.359,E4 +0.000} C_DIS
LIN {X -153.552,Y +1158.113,Z +0.000,A -20.000,E1 -11.113,E3 +68736.110,E4 +0.000} C_DIS
LIN {X -156.311,Y +1155.540,Z +0.000,A -20.000,E1 -0.839,E3 +68779.470,E4 +0.000} C_DIS
LIN {X -161.281,Y +1151.851,Z +0.000,A -20.000,E1 +7.737,E3 +68809.369,E4 +0.000} C_DIS
LIN {X -167.493,Y +1147.157,Z +0.000,A -20.000,E1 +16.195,E3 +68833.808,E4 +0.000} C_DIS
LIN {X -173.235,Y +1142.221,Z +0.000,A -20.000,E1 +22.930,E3 +68851.110,E4 +0.000} C_DIS
LIN {X -181.123,Y +1133.734,Z +0.000,A -20.000,E1 +30.868,E3 +68871.866,E4 +0.000} C_DIS
LIN {X -189.654,Y +1120.856,Z +0.000,A -20.000,E1 +39.018,E3 +68893.880,E4 +0.000} C_DIS
LIN {X -195.246,Y +1107.046,Z +0.000,A -20.000,E1 +44.515,E3 +68911.782,E4 +0.000} C_DIS
LIN {X -198.051,Y +1092.368,Z +0.000,A -20.000,E1 +47.947,E3 +68928.308,E4 +0.000} C_DIS
LIN {X -198.143,Y +1081.370,Z +0.000,A -19.806,E1 +49.153,E3 +68940.169,E4 +0.000} C_DIS
LIN {X -197.177,Y +1073.569,Z +0.000,A -17.356,E1 +49.162,E3 +68948.753,E4 +0.000} C_DIS
LIN {X -195.448,Y +1066.139,Z +0.000,A -12.154,E1 +48.512,E3 +68957.348,E4 +0.000} C_DIS
LIN {X -193.346,Y +1058.941,Z +0.000,A -7.133,E1 +47.724,E3 +68966.228,E4 +0.000} C_DIS
LIN {X -191.781,Y +1050.839,Z +0.000,A -3.715,E1 +47.274,E3 +68976.561,E4 +0.000} C_DIS
LIN {X -190.795,Y +1039.355,Z +0.000,A -0.983,E1 +46.842,E3 +68991.221,E4 +0.000} C_DIS
LIN {X -190.395,Y +1028.856,Z +0.000,A -0.089,E1 +46.598,E3 +69004.615,E4 +0.000} C_DIS
LIN {X -190.239,Y +1018.851,Z +0.000,A -0.004,E1 +46.529,E3 +69017.383,E4 +0.000} C_DIS
LIN {X -190.161,Y +1004.975,Z +0.000,A +0.000,E1 +46.506,E3 +69035.097,E4 +0.000} C_DIS
LIN {X -190.142,Y +412.853,Z +0.000,A +0.000,E1 +46.501,E3 +69791.303,E4 +0.000} C_DIS
LIN {X -190.147,Y +401.077,Z +0.000,A +0.000,E1 +46.499,E3 +69806.344,E4 +0.000} C_DIS
LIN {X -190.159,Y +390.929,Z +0.000,A +0.000,E1 +46.494,E3 +69819.310,E4 +0.000} C_DIS
LIN {X -190.174,Y +383.973,Z +0.000,A +0.000,E1 +46.484,E3 +69828.203,E4 +0.000} C_DIS
LIN {X -190.200,Y +373.815,Z +0.000,A +0.000,E1 +46.448,E3 +69841.208,E4 +0.000} C_DIS
LIN {X -190.154,Y +361.003,Z +0.000,A +0.000,E1 +46.303,E3 +69857.702,E4 +0.000} C_DIS
LIN {X -189.772,Y +350.660,Z +0.000,A +0.049,E1 +45.996,E3 +69871.241,E4 +0.000} C_DIS
LIN {X -189.325,Y +346.917,Z +0.000,A +0.243,E1 +45.771,E3 +69876.310,E4 +0.000} C_DIS
LIN {X -188.196,Y +342.754,Z +0.000,A +1.966,E1 +45.249,E3 +69882.318,E4 +0.000} C_DIS
LIN {X -185.199,Y +337.023,Z +0.000,A +6.630,E1 +43.793,E3 +69891.692,E4 +0.000} C_DIS
LIN {X -181.141,Y +331.596,Z +0.000,A +12.274,E1 +41.569,E3 +69902.252,E4 +0.000} C_DIS
LIN {X -176.762,Y +326.804,Z +0.000,A +17.560,E1 +38.898,E3 +69913.676,E4 +0.000} C_DIS
LIN {X -172.184,Y +322.578,Z +0.000,A +19.859,E1 +36.197,E3 +69926.406,E4 +0.000} C_DIS
LIN {X -165.998,Y +317.874,Z +0.000,A +20.000,E1 +32.027,E3 +69946.164,E4 +0.000} C_DIS
LIN {X -160.137,Y +314.334,Z +0.000,A +20.000,E1 +26.368,E3 +69970.533,E4 +0.000} C_DIS
LIN {X -155.624,Y +312.245,Z +0.000,A +20.000,E1 +19.506,E3 +69999.209,E4 +0.000} C_DIS
LIN {X -153.557,Y +311.879,Z +0.000,A +20.000,E1 +11.113,E3 +70034.964,E4 +0.000} C_DIS
LIN {X -155.320,Y +313.348,Z +0.000,A +20.000,E1 +3.401,E3 +70068.148,E4 +0.000} C_DIS
LIN {X -160.005,Y +315.804,Z +0.000,A +20.000,E1 -4.720,E3 +70098.526,E4 +0.000} C_DIS
LIN {X -164.504,Y +318.255,Z +0.000,A +20.000,E1 -10.663,E3 +70117.895,E4 +0.000} C_DIS
LIN {X -170.340,Y +322.684,Z +0.000,A +20.000,E1 -17.457,E3 +70137.927,E4 +0.000} C_DIS
LIN {X -175.568,Y +329.106,Z +0.000,A +20.000,E1 -24.747,E3 +70155.161,E4 +0.000} C_DIS
LIN {X -184.074,Y +340.065,Z +0.000,A +20.000,E1 -33.664,E3 +70178.101,E4 +0.000} C_DIS
LIN {X -190.779,Y +351.388,Z +0.000,A +20.000,E1 -40.083,E3 +70195.879,E4 +0.000} C_DIS
LIN {X -195.254,Y +362.955,Z +0.000,A +20.000,E1 -44.515,E3 +70210.632,E4 +0.000} C_DIS
LIN {X -197.754,Y +374.780,Z +0.000,A +20.000,E1 -47.450,E3 +70224.054,E4 +0.000} C_DIS
LIN {X -198.310,Y +383.215,Z +0.000,A +19.956,E1 -48.698,E3 +70233.178,E4 +0.000} C_DIS
LIN {X -197.912,Y +391.275,Z +0.000,A +18.601,E1 -49.158,E3 +70241.896,E4 +0.000} C_DIS
LIN {X -196.679,Y +398.944,Z +0.000,A +13.989,E1 -48.784,E3 +70250.450,E4 +0.000} C_DIS
LIN {X -194.742,Y +406.288,Z +0.000,A +8.476,E1 -48.001,E3 +70259.133,E4 +0.000} C_DIS
LIN {X -192.748,Y +413.472,Z +0.000,A +3.905,E1 -47.267,E3 +70268.143,E4 +0.000} C_DIS
LIN {X -191.781,Y +419.162,Z +0.000,A +1.739,E1 -46.975,E3 +70275.411,E4 +0.000} C_DIS
LIN {X -190.795,Y +430.646,Z +0.000,A +0.152,E1 -46.707,E3 +70290.072,E4 +0.000} C_DIS
LIN {X -190.395,Y +441.145,Z +0.000,A +0.001,E1 -46.583,E3 +70303.465,E4 +0.000} C_DIS
LIN {X -190.239,Y +451.150,Z +0.000,A -0.000,E1 -46.528,E3 +70316.233,E4 +0.000} C_DIS
LIN {X -190.161,Y +465.026,Z +0.000,A -0.000,E1 -46.506,E3 +70333.948,E4 +0.000} C_DIS
LIN {X -190.142,Y +1057.148,Z +0.000,A -0.000,E1 -46.500,E3 +71090.154,E4 +0.000} C_DIS
LIN {X -190.147,Y +1068.924,Z +0.000,A -0.000,E1 -46.499,E3 +71105.195,E4 +0.000} C_DIS
LIN {X -190.159,Y +1079.072,Z +0.000,A -0.000,E1 -46.493,E3 +71118.160,E4 +0.000} C_DIS
LIN {X -190.174,Y +1086.028,Z +0.000,A -0.000,E1 -46.483,E3 +71127.054,E4 +0.000} C_DIS
LIN {X -190.200,Y +1096.186,Z +0.000,A -0.000,E1 -46.448,E3 +71140.058,E4 +0.000} C_DIS
LIN {X -190.154,Y +1108.998,Z +0.000,A -0.054,E1 -46.295,E3 +71156.553,E4 +0.000} C_DIS
LIN {X -189.772,Y +1119.341,Z +0.000,A -0.752,E1 -45.902,E3 +71170.091,E4 +0.000} C_DIS
LIN {X -189.097,Y +1124.276,Z +0.000,A -2.508,E1 -45.397,E3 +71176.823,E4 +0.000} C_DIS
LIN {X -187.410,Y +1129.069,Z +0.000,A -5.304,E1 -44.585,E3 +71183.996,E4 +0.000} C_DIS
LIN {X -183.899,Y +1134.873,Z +0.000,A -10.372,E1 -42.805,E3 +71194.002,E4 +0.000} C_DIS
LIN {X -179.711,Y +1140.065,Z +0.000,A -15.940,E1 -40.393,E3 +71204.788,E4 +0.000} C_DIS
LIN {X -176.763,Y +1143.197,Z +0.000,A -18.748,E1 -38.674,E3 +71212.526,E4 +0.000} C_DIS
LIN {X -172.185,Y +1147.423,Z +0.000,A -19.971,E1 -36.175,E3 +71225.256,E4 +0.000} C_DIS
LIN {X -165.999,Y +1152.127,Z +0.000,A -20.000,E1 -32.027,E3 +71245.014,E4 +0.000} C_DIS
LIN {X -160.138,Y +1155.667,Z +0.000,A -20.000,E1 -26.368,E3 +71269.384,E4 +0.000} C_DIS
LIN {X -155.625,Y +1157.756,Z +0.000,A -20.000,E1 -19.505,E3 +71298.060,E4 +0.000} C_DIS
LIN {X -153.552,Y +1158.113,Z +0.000,A -20.000,E1 -11.113,E3 +71333.811,E4 +0.000} C_DIS
LIN {X -156.311,Y +1155.540,Z +0.000,A -20.000,E1 -0.839,E3 +71377.171,E4 +0.000} C_DIS
LIN {X -161.281,Y +1151.851,Z +0.000,A -20.000,E1 +7.737,E3 +71407.070,E4 +0.000} C_DIS
LIN {X -167.493,Y +1147.157,Z +0.000,A -20.000,E1 +16.195,E3 +71431.509,E4 +0.000} C_DIS
LIN {X -173.235,Y +1142.221,Z +0.000,A -20.000,E1 +22.930,E3 +71448.811,E4 +0.000} C_DIS
LIN {X -181.123,Y +1133.734,Z +0.000,A -20.000,E1 +30.868,E3 +71469.567,E4 +0.000} C_DIS
LIN {X -189.654,Y +1120.856,Z +0.000,A -20.000,E1 +39.018,E3 +71491.581,E4 +0.000} C_DIS
LIN {X -195.246,Y +1107.046,Z +0.000,A -20.000,E1 +44.515,E3 +71509.483,E4 +0.000} C_DIS
LIN {X -198.051,Y +1092.368,Z +0.000,A -20.000,E1 +47.947,E3 +71526.009,E4 +0.000} C_DIS
LIN {X -198.143,Y +1081.370,Z +0.000,A -19.806,E1 +49.153,E3 +71537.870,E4 +0.000} C_DIS
LIN {X -197.177,Y +1073.569,Z +0.000,A -17.356,E1 +49.162,E3 +71546.454,E4 +0.000} C_DIS
LIN {X -195.448,Y +1066.139,Z +0.000,A -12.154,E1 +48.512,E3 +71555.049,E4 +0.000} C_DIS
LIN {X -193.346,Y +1058.941,Z +0.000,A -7.133,E1 +47.724,E3 +71563.929,E4 +0.000} C_DIS
LIN {X -191.781,Y +1050.839,Z +0.000,A -3.715,E1 +47.274,E3 +71574.262,E4 +0.000} C_DIS
LIN {X -190.795,Y +1039.355,Z +0.000,A -0.983,E1 +46.842,E3 +71588.922,E4 +0.000} C_DIS
LIN {X -190.395,Y +1028.856,Z +0.000,A -0.089,E1 +46.598,E3 +71602.316,E4 +0.000} C_DIS
LIN {X -190.239,Y +1018.851,Z +0.000,A -0.004,E1 +46.529,E3 +71615.084,E4 +0.000} C_DIS
LIN {X -190.161,Y +1004.975,Z +0.000,A +0.000,E1 +46.506,E3 +71632.798,E4 +0.000} C_DIS
LIN {X -190.142,Y +412.853,Z +0.000,A +0.000,E1 +46.501,E3 +72389.004,E4 +0.000} C_DIS
LIN {X -190.147,Y +401.077,Z +0.000,A +0.000,E1 +46.499,E3 +72404.045,E4 +0.000} C_DIS
LIN {X -190.159,Y +390.929,Z +0.000,A +0.000,E1 +46.494,E3 +72417.011,E4 +0.000} C_DIS
LIN {X -190.174,Y +383.973,Z +0.000,A +0.000,E1 +46.484,E3 +72425.904,E4 +0.000} C_DIS
LIN {X -190.200,Y +373.815,Z +0.000,A +0.000,E1 +46.448,E3 +72438.909,E4 +0.000} C_DIS
LIN {X -190.154,Y +361.003,Z +0.000,A +0.000,E1 +46.303,E3 +72455.403,E4 +0.000} C_DIS
LIN {X -189.772,Y +350.660,Z +0.000,A +0.049,E1 +45.996,E3 +72468.942,E4 +0.000} C_DIS
LIN {X -189.325,Y +346.917,Z +0.000,A +0.243,E1 +45.771,E3 +72474.011,E4 +0.000} C_DIS
LIN {X -188.196,Y +342.754,Z +0.000,A +1.966,E1 +45.249,E3 +72480.019,E4 +0.000} C_DIS
LIN {X -185.199,Y +337.023,Z +0.000,A +6.630,E1 +43.793,E3 +72489.393,E4 +0.000} C_DIS
LIN {X -181.141,Y +331.596,Z +0.000,A +12.274,E1 +41.569,E3 +72499.953,E4 +0.000} C_DIS
LIN {X -176.762,Y +326.804,Z +0.000,A +17.560,E1 +38.898,E3 +72511.377,E4 +0.000} C_DIS
LIN {X -172.184,Y +322.578,Z +0.000,A +19.859,E1 +36.197,E3 +72524.107,E4 +0.000} C_DIS
LIN {X -165.998,Y +317.874,Z +0.000,A +20.000,E1 +32.027,E3 +72543.865,E4 +0.000} C_DIS
LIN {X -160.137,Y +314.334,Z +0.000,A +20.000,E1 +26.368,E3 +72568.234,E4 +0.000} C_DIS
LIN {X -155.624,Y +312.245,Z +0.000,A +20.000,E1 +19.506,E3 +72596.910,E4 +0.000} C_DIS
LIN {X -153.557,Y +311.879,Z +0.000,A +20.000,E1 +11.113,E3 +72632.665,E4 +0.000} C_DIS
LIN {X -155.320,Y +313.348,Z +0.000,A +20.000,E1 +3.401,E3 +72665.849,E4 +0.000} C_DIS
LIN {X -160.005,Y +315.804,Z +0.000,A +20.000,E1 -4.720,E3 +72696.227,E4 +0.000} C_DIS
LIN {X -164.504,Y +318.255,Z +0.000,A +20.000,E1 -10.663,E3 +72715.596,E4 +0.000} C_DIS
LIN {X -170.340,Y +322.684,Z +0.000,A +20.000,E1 -17.457,E3 +72735.628,E4 +0.000} C_DIS
LIN {X -175.568,Y +329.106,Z +0.000,A +20.000,E1 -24.747,E3 +72752.862,E4 +0.000} C_DIS
LIN {X -184.074,Y +340.065,Z +0.000,A +20.000,E1 -33.664,E3 +72775.802,E4 +0.000} C_DIS
LIN {X -190.779,Y +351.388,Z +0.000,A +20.000,E1 -40.083,E3 +72793.580,E4 +0.000} C_DIS
LIN {X -195.254,Y +362.955,Z +0.000,A +20.000,E1 -44.515,E3 +72808.333,E4 +0.000} C_DIS
LIN {X -197.754,Y +374.780,Z +0.000,A +20.000,E1 -47.450,E3 +72821.755,E4 +0.000} C_DIS
LIN {X -198.310,Y +383.215,Z +0.000,A +19.956,E1 -48.698,E3 +72830.879,E4 +0.000} C_DIS
LIN {X -197.912,Y +391.275,Z +0.000,A +18.601,E1 -49.158,E3 +72839.597,E4 +0.000} C_DIS
LIN {X -196.679,Y +398.944,Z +0.000,A +13.989,E1 -48.784,E3 +72848.151,E4 +0.000} C_DIS
LIN {X -194.742,Y +406.288,Z +0.000,A +8.476,E1 -48.001,E3 +72856.834,E4 +0.000} C_DIS
LIN {X -192.748,Y +413.472,Z +0.000,A +3.905,E1 -47.267,E3 +72865.844,E4 +0.000} C_DIS
LIN {X -191.781,Y +419.162,Z +0.000,A +1.739,E1 -46.975,E3 +72873.112,E4 +0.000} C_DIS
LIN {X -190.795,Y +430.646,Z +0.000,A +0.152,E1 -46.707,E3 +72887.773,E4 +0.000} C_DIS
LIN {X -190.395,Y +441.145,Z +0.000,A +0.001,E1 -46.583,E3 +72901.166,E4 +0.000} C_DIS
LIN {X -190.239,Y +451.150,Z +0.000,A -0.000,E1 -46.528,E3 +72913.934,E4 +0.000} C_DIS
LIN {X -190.161,Y +465.026,Z +0.000,A -0.000,E1 -46.506,E3 +72931.649,E4 +0.000} C_DIS
LIN {X -190.142,Y +1057.148,Z +0.000,A -0.000,E1 -46.500,E3 +73687.855,E4 +0.000} C_DIS
LIN {X -190.147,Y +1068.924,Z +0.000,A -0.000,E1 -46.499,E3 +73702.896,E4 +0.000} C_DIS
LIN {X -190.159,Y +1079.072,Z +0.000,A -0.000,E1 -46.493,E3 +73715.861,E4 +0.000} C_DIS
LIN {X -190.174,Y +1086.028,Z +0.000,A -0.000,E1 -46.483,E3 +73724.755,E4 +0.000} C_DIS
LIN {X -190.200,Y +1096.186,Z +0.000,A -0.000,E1 -46.448,E3 +73737.759,E4 +0.000} C_DIS
LIN {X -190.154,Y +1108.998,Z +0.000,A -0.054,E1 -46.295,E3 +73754.254,E4 +0.000} C_DIS
LIN {X -189.772,Y +1119.341,Z +0.000,A -0.752,E1 -45.902,E3 +73767.792,E4 +0.000} C_DIS
LIN {X -189.097,Y +1124.276,Z +0.000,A -2.508,E1 -45.397,E3 +73774.524,E4 +0.000} C_DIS
LIN {X -187.410,Y +1129.069,Z +0.000,A -5.304,E1 -44.585,E3 +73781.697,E4 +0.000} C_DIS
LIN {X -183.899,Y +1134.873,Z +0.000,A -10.372,E1 -42.805,E3 +73791.703,E4 +0.000} C_DIS
LIN {X -179.711,Y +1140.065,Z +0.000,A -15.940,E1 -40.393,E3 +73802.489,E4 +0.000} C_DIS
LIN {X -176.763,Y +1143.197,Z +0.000,A -18.748,E1 -38.674,E3 +73810.227,E4 +0.000} C_DIS
LIN {X -172.185,Y +1147.423,Z +0.000,A -19.971,E1 -36.175,E3 +73822.957,E4 +0.000} C_DIS
LIN {X -165.999,Y +1152.127,Z +0.000,A -20.000,E1 -32.027,E3 +73842.715,E4 +0.000} C_DIS
LIN {X -160.138,Y +1155.667,Z +0.000,A -20.000,E1 -26.368,E3 +73867.085,E4 +0.000} C_DIS
LIN {X -155.625,Y +1157.756,Z +0.000,A -20.000,E1 -19.505,E3 +73895.761,E4 +0.000} C_DIS
LIN {X -153.552,Y +1158.113,Z +0.000,A -20.000,E1 -11.113,E3 +73931.512,E4 +0.000} C_DIS
LIN {X -156.311,Y +1155.540,Z +0.000,A -20.000,E1 -0.839,E3 +73974.872,E4 +0.000} C_DIS
LIN {X -161.281,Y +1151.851,Z +0.000,A -20.000,E1 +7.737,E3 +74004.771,E4 +0.000} C_DIS
LIN {X -167.493,Y +1147.157,Z +0.000,A -20.000,E1 +16.195,E3 +74029.210,E4 +0.000} C_DIS
LIN {X -173.235,Y +1142.221,Z +0.000,A -20.000,E1 +22.930,E3 +74046.512,E4 +0.000} C_DIS
LIN {X -181.123,Y +1133.734,Z +0.000,A -20.000,E1 +30.868,E3 +74067.268,E4 +0.000} C_DIS
LIN {X -189.654,Y +1120.856,Z +0.000,A -20.000,E1 +39.018,E3 +74089.282,E4 +0.000} C_DIS
LIN {X -195.246,Y +1107.046,Z +0.000,A -20.000,E1 +44.515,E3 +74107.184,E4 +0.000} C_DIS
LIN {X -198.051,Y +1092.368,Z +0.000,A -20.000,E1 +47.947,E3 +74123.710,E4 +0.000} C_DIS
LIN {X -198.143,Y +1081.370,Z +0.000,A -19.806,E1 +49.153,E3 +74135.571,E4 +0.000} C_DIS
LIN {X -197.177,Y +1073.569,Z +0.000,A -17.356,E1 +49.162,E3 +74144.155,E4 +0.000} C_DIS
LIN {X -195.448,Y +1066.139,Z +0.000,A -12.154,E1 +48.512,E3 +74152.750,E4 +0.000} C_DIS
LIN {X -193.346,Y +1058.941,Z +0.000,A -7.133,E1 +47.724,E3 +74161.630,E4 +0.000} C_DIS
LIN {X -191.781,Y +1050.839,Z +0.000,A -3.715,E1 +47.274,E3 +74171.963,E4 +0.000} C_DIS
LIN {X -190.795,Y +1039.355,Z +0.000,A -0.983,E1 +46.842,E3 +74186.623,E4 +0.000} C_DIS
LIN {X -190.395,Y +1028.856,Z +0.000,A -0.089,E1 +46.598,E3 +74200.017,E4 +0.000} C_DIS
LIN {X -190.239,Y +1018.851,Z +0.000,A -0.004,E1 +46.529,E3 +74212.785,E4 +0.000} C_DIS
LIN {X -190.161,Y +1004.975,Z +0.000,A +0.000,E1 +46.506,E3 +74230.499,E4 +0.000} C_DIS
LIN {X -190.142,Y +412.853,Z +0.000,A +0.000,E1 +46.501,E3 +74986.705,E4 +0.000} C_DIS
LIN {X -190.147,Y +401.077,Z +0.000,A +0.000,E1 +46.499,E3 +75001.746,E4 +0.000} C_DIS
LIN {X -190.159,Y +390.929,Z +0.000,A +0.000,E1 +46.494,E3 +75014.712,E4 +0.000} C_DIS
LIN {X -190.174,Y +383.973,Z +0.000,A +0.000,E1 +46.484,E3 +75023.605,E4 +0.000} C_DIS
LIN {X -190.200,Y +373.815,Z +0.000,A +0.000,E1 +46.448,E3 +75036.610,E4 +0.000} C_DIS
LIN {X -190.154,Y +361.003,Z +0.000,A +0.000,E1 +46.303,E3 +75053.104,E4 +0.000} C_DIS
LIN {X -189.772,Y +350.660,Z +0.000,A +0.049,E1 +45.996,E3 +75066.643,E4 +0.000} C_DIS
LIN {X -189.325,Y +346.917,Z +0.000,A +0.243,E1 +45.771,E3 +75071.712,E4 +0.000} C_DIS
LIN {X -188.196,Y +342.754,Z +0.000,A +1.966,E1 +45.249,E3 +75077.720,E4 +0.000} C_DIS
LIN {X -185.199,Y +337.023,Z +0.000,A +6.630,E1 +43.793,E3 +75087.094,E4 +0.000} C_DIS
LIN {X -181.141,Y +331.596,Z +0.000,A +12.274,E1 +41.569,E3 +75097.654,E4 +0.000} C_DIS
LIN {X -176.762,Y +326.804,Z +0.000,A +17.560,E1 +38.898,E3 +75109.078,E4 +0.000} C_DIS
LIN {X -172.184,Y +322.578,Z +0.000,A +19.859,E1 +36.197,E3 +75121.808,E4 +0.000} C_DIS
LIN {X -165.998,Y +317.874,Z +0.000,A +20.000,E1 +32.027,E3 +75141.566,E4 +0.000} C_DIS
LIN {X -160.137,Y +314.334,Z +0.000,A +20.000,E1 +26.368,E3 +75165.935,E4 +0.000} C_DIS
LIN {X -155.624,Y +312.245,Z +0.000,A +20.000,E1 +19.506,E3 +75194.611,E4 +0.000} C_DIS
LIN {X -153.557,Y +311.879,Z +0.000,A +20.000,E1 +11.113,E3 +75230.366,E4 +0.000} C_DIS
LIN {X -155.320,Y +313.348,Z +0.000,A +20.000,E1 +3.401,E3 +75263.550,E4 +0.000} C_DIS
LIN {X -160.005,Y +315.804,Z +0.000,A +20.000,E1 -4.720,E3 +75293.928,E4 +0.000} C_DIS
LIN {X -164.504,Y +318.255,Z +0.000,A +20.000,E1 -10.663,E3 +75313.297,E4 +0.000} C_DIS
LIN {X -170.340,Y +322.684,Z +0.000,A +20.000,E1 -17.457,E3 +75333.329,E4 +0.000} C_DIS
LIN {X -175.568,Y +329.106,Z +0.000,A +20.000,E1 -24.747,E3 +75350.563,E4 +0.000} C_DIS
LIN {X -184.074,Y +340.065,Z +0.000,A +20.000,E1 -33.664,E3 +75373.503,E4 +0.000} C_DIS
LIN {X -190.779,Y +351.388,Z +0.000,A +20.000,E1 -40.083,E3 +75391.281,E4 +0.000} C_DIS
LIN {X -195.254,Y +362.955,Z +0.000,A +20.000,E1 -44.515,E3 +75406.034,E4 +0.000} C_DIS
LIN {X -197.754,Y +374.780,Z +0.000,A +20.000,E1 -47.450,E3 +75419.456,E4 +0.000} C_DIS
LIN {X -198.310,Y +383.215,Z +0.000,A +19.956,E1 -48.698,E3 +75428.580,E4 +0.000} C_DIS
LIN {X -197.912,Y +391.275,Z +0.000,A +18.601,E1 -49.158,E3 +75437.298,E4 +0.000} C_DIS
LIN {X -196.679,Y +398.944,Z +0.000,A +13.989,E1 -48.784,E3 +75445.852,E4 +0.000} C_DIS
LIN {X -194.742,Y +406.288,Z +0.000,A +8.476,E1 -48.001,E3 +75454.535,E4 +0.000} C_DIS
LIN {X -192.748,Y +413.472,Z +0.000,A +3.905,E1 -47.267,E3 +75463.545,E4 +0.000} C_DIS
LIN {X -191.781,Y +419.162,Z +0.000,A +1.739,E1 -46.975,E3 +75470.813,E4 +0.000} C_DIS
LIN {X -190.795,Y +430.646,Z +0.000,A +0.152,E1 -46.707,E3 +75485.474,E4 +0.000} C_DIS
LIN {X -190.395,Y +441.145,Z +0.000,A +0.001,E1 -46.583,E3 +75498.867,E4 +0.000} C_DIS
LIN {X -190.239,Y +451.150,Z +0.000,A -0.000,E1 -46.528,E3 +75511.635,E4 +0.000} C_DIS
LIN {X -190.161,Y +465.026,Z +0.000,A -0.000,E1 -46.506,E3 +75529.350,E4 +0.000} C_DIS
LIN {X -190.142,Y +1057.148,Z +0.000,A -0.000,E1 -46.500,E3 +76285.556,E4 +0.000} C_DIS
LIN {X -190.147,Y +1068.924,Z +0.000,A -0.000,E1 -46.499,E3 +76300.597,E4 +0.000} C_DIS
LIN {X -190.159,Y +1079.072,Z +0.000,A -0.000,E1 -46.493,E3 +76313.562,E4 +0.000} C_DIS
LIN {X -190.174,Y +1086.028,Z +0.000,A -0.000,E1 -46.483,E3 +76322.456,E4 +0.000} C_DIS
LIN {X -190.200,Y +1096.186,Z +0.000,A -0.000,E1 -46.448,E3 +76335.460,E4 +0.000} C_DIS
LIN {X -190.154,Y +1108.998,Z +0.000,A -0.054,E1 -46.295,E3 +76351.955,E4 +0.000} C_DIS
LIN {X -189.772,Y +1119.341,Z +0.000,A -0.752,E1 -45.902,E3 +76365.493,E4 +0.000} C_DIS
LIN {X -189.097,Y +1124.276,Z +0.000,A -2.508,E1 -45.397,E3 +76372.225,E4 +0.000} C_DIS
LIN {X -187.410,Y +1129.069,Z +0.000,A -5.304,E1 -44.585,E3 +76379.398,E4 +0.000} C_DIS
LIN {X -183.899,Y +1134.873,Z +0.000,A -10.372,E1 -42.805,E3 +76389.404,E4 +0.000} C_DIS
LIN {X -179.711,Y +1140.065,Z +0.000,A -15.940,E1 -40.393,E3 +76400.190,E4 +0.000} C_DIS
LIN {X -176.763,Y +1143.197,Z +0.000,A -18.748,E1 -38.674,E3 +76407.928,E4 +0.000} C_DIS
LIN {X -172.185,Y +1147.423,Z +0.000,A -19.971,E1 -36.175,E3 +76420.658,E4 +0.000} C_DIS
LIN {X -165.999,Y +1152.127,Z +0.000,A -20.000,E1 -32.027,E3 +76440.416,E4 +0.000} C_DIS
LIN {X -160.138,Y +1155.667,Z +0.000,A -20.000,E1 -26.368,E3 +76464.786,E4 +0.000} C_DIS
LIN {X -155.625,Y +1157.756,Z +0.000,A -20.000,E1 -19.505,E3 +76493.462,E4 +0.000} C_DIS
LIN {X -153.552,Y +1158.113,Z +0.000,A -20.000,E1 -11.113,E3 +76529.213,E4 +0.000} C_DIS
LIN {X -156.311,Y +1155.540,Z +0.000,A -20.000,E1 -0.839,E3 +76572.573,E4 +0.000} C_DIS
LIN {X -161.281,Y +1151.851,Z +0.000,A -20.000,E1 +7.737,E3 +76602.472,E4 +0.000} C_DIS
LIN {X -167.493,Y +1147.157,Z +0.000,A -20.000,E1 +16.195,E3 +76626.911,E4 +0.000} C_DIS
LIN {X -173.235,Y +1142.221,Z +0.000,A -20.000,E1 +22.930,E3 +76644.213,E4 +0.000} C_DIS
LIN {X -181.123,Y +1133.734,Z +0.000,A -20.000,E1 +30.868,E3 +76664.969,E4 +0.000} C_DIS
LIN {X -189.654,Y +1120.856,Z +0.000,A -20.000,E1 +39.018,E3 +76686.983,E4 +0.000} C_DIS
LIN {X -195.246,Y +1107.046,Z +0.000,A -20.000,E1 +44.515,E3 +76704.885,E4 +0.000} C_DIS
LIN {X -198.051,Y +1092.368,Z +0.000,A -20.000,E1 +47.947,E3 +76721.411,E4 +0.000} C_DIS
LIN {X -198.143,Y +1081.370,Z +0.000,A -19.806,E1 +49.153,E3 +76733.272,E4 +0.000} C_DIS
LIN {X -197.177,Y +1073.569,Z +0.000,A -17.356,E1 +49.162,E3 +76741.856,E4 +0.000} C_DIS
LIN {X -195.448,Y +1066.139,Z +0.000,A -12.154,E1 +48.512,E3 +76750.451,E4 +0.000} C_DIS
LIN {X -193.346,Y +1058.941,Z +0.000,A -7.133,E1 +47.724,E3 +76759.331,E4 +0.000} C_DIS
LIN {X -191.781,Y +1050.839,Z +0.000,A -3.715,E1 +47.274,E3 +76769.664,E4 +0.000} C_DIS
LIN {X -190.795,Y +1039.355,Z +0.000,A -0.983,E1 +46.842,E3 +76784.324,E4 +0.000} C_DIS
LIN {X -190.395,Y +1028.856,Z +0.000,A -0.089,E1 +46.598,E3 +76797.718,E4 +0.000} C_DIS
LIN {X -190.239,Y +1018.851,Z +0.000,A -0.004,E1 +46.529,E3 +76810.486,E4 +0.000} C_DIS
LIN {X -190.161,Y +1004.975,Z +0.000,A +0.000,E1 +46.506,E3 +76828.200,E4 +0.000} C_DIS
LIN {X -190.142,Y +412.853,Z +0.000,A +0.000,E1 +46.501,E3 +77584.406,E4 +0.000} C_DIS
LIN {X -190.147,Y +401.077,Z +0.000,A +0.000,E1 +46.499,E3 +77599.447,E4 +0.000} C_DIS
LIN {X -190.159,Y +390.929,Z +0.000,A +0.000,E1 +46.494,E3 +77612.413,E4 +0.000} C_DIS
LIN {X -190.174,Y +383.973,Z +0.000,A +0.000,E1 +46.484,E3 +77621.306,E4 +0.000} C_DIS
LIN {X -190.200,Y +373.815,Z +0.000,A +0.000,E1 +46.448,E3 +77634.311,E4 +0.000} C_DIS
LIN {X -190.154,Y +361.003,Z +0.000,A +0.000,E1 +46.303,E3 +77650.805,E4 +0.000} C_DIS
LIN {X -189.772,Y +350.660,Z +0.000,A +0.049,E1 +45.996,E3 +77664.344,E4 +0.000} C_DIS
LIN {X -189.325,Y +346.917,Z +0.000,A +0.243,E1 +45.771,E3 +77669.413,E4 +0.000} C_DIS
LIN {X -188.196,Y +342.754,Z +0.000,A +1.966,E1 +45.249,E3 +77675.421,E4 +0.000} C_DIS
LIN {X -185.199,Y +337.023,Z +0.000,A +6.630,E1 +43.793,E3 +77684.795,E4 +0.000} C_DIS
LIN {X -181.141,Y +331.596,Z +0.000,A +12.274,E1 +41.569,E3 +77695.355,E4 +0.000} C_DIS
LIN {X -176.762,Y +326.804,Z +0.000,A +17.560,E1 +38.898,E3 +77706.779,E4 +0.000} C_DIS
LIN {X -172.184,Y +322.578,Z +0.000,A +19.859,E1 +36.197,E3 +77719.509,E4 +0.000} C_DIS
LIN {X -165.998,Y +317.874,Z +0.000,A +20.000,E1 +32.027,E3 +77739.267,E4 +0.000} C_DIS
LIN {X -160.137,Y +314.334,Z +0.000,A +20.000,E1 +26.368,E3 +77763.636,E4 +0.000} C_DIS
LIN {X -155.624,Y +312.245,Z +0.000,A +20.000,E1 +19.506,E3 +77792.312,E4 +0.000} C_DIS
LIN {X -153.557,Y +311.879,Z +0.000,A +20.000,E1 +11.113,E3 +77828.067,E4 +0.000} C_DIS
LIN {X -155.320,Y +313.348,Z +0.000,A +20.000,E1 +3.401,E3 +77861.251,E4 +0.000} C_DIS
LIN {X -160.005,Y +315.804,Z +0.000,A +20.000,E1 -4.720,E3 +77891.629,E4 +0.000} C_DIS
LIN {X -164.504,Y +318.255,Z +0.000,A +20.000,E1 -10.663,E3 +77910.998,E4 +0.000} C_DIS
LIN {X -170.340,Y +322.684,Z +0.000,A +20.000,E1 -17.457,E3 +77931.030,E4 +0.000} C_DIS
LIN {X -175.568,Y +329.106,Z +0.000,A +20.000,E1 -24.747,E3 +77948.264,E4 +0.000} C_DIS
LIN {X -184.074,Y +340.065,Z +0.000,A +20.000,E1 -33.664,E3 +77971.204,E4 +0.000} C_DIS
LIN {X -190.779,Y +351.388,Z +0.000,A +20.000,E1 -40.083,E3 +77988.982,E4 +0.000} C_DIS
LIN {X -195.254,Y +362.955,Z +0.000,A +20.000,E1 -44.515,E3 +78003.735,E4 +0.000} C_DIS
LIN {X -197.754,Y +374.780,Z +0.000,A +20.000,E1 -47.450,E3 +78017.157,E4 +0.000} C_DIS
LIN {X -198.310,Y +383.215,Z +0.000,A +19.956,E1 -48.698,E3 +78026.281,E4 +0.000} C_DIS
LIN {X -197.912,Y +391.275,Z +0.000,A +18.601,E1 -49.158,E3 +78034.999,E4 +0.000} C_DIS
LIN {X -196.679,Y +398.944,Z +0.000,A +13.989,E1 -48.784,E3 +78043.553,E4 +0.000} C_DIS
LIN {X -194.742,Y +406.288,Z +0.000,A +8.476,E1 -48.001,E3 +78052.236,E4 +0.000} C_DIS
LIN {X -192.748,Y +413.472,Z +0.000,A +3.905,E1 -47.267,E3 +78061.246,E4 +0.000} C_DIS
LIN {X -191.781,Y +419.162,Z +0.000,A +1.739,E1 -46.975,E3 +78068.514,E4 +0.000} C_DIS
LIN {X -190.795,Y +430.646,Z +0.000,A +0.152,E1 -46.707,E3 +78083.175,E4 +0.000} C_DIS
LIN {X -190.395,Y +441.145,Z +0.000,A +0.001,E1 -46.583,E3 +78096.568,E4 +0.000} C_DIS
LIN {X -190.239,Y +451.150,Z +0.000,A -0.000,E1 -46.528,E3 +78109.336,E4 +0.000} C_DIS
LIN {X -190.161,Y +465.026,Z +0.000,A -0.000,E1 -46.506,E3 +78127.051,E4 +0.000} C_DIS
LIN {X -190.142,Y +1057.148,Z +0.000,A -0.000,E1 -46.500,E3 +78883.257,E4 +0.000} C_DIS
LIN {X -190.147,Y +1068.924,Z +0.000,A -0.000,E1 -46.499,E3 +78898.298,E4 +0.000} C_DIS
LIN {X -190.159,Y +1079.072,Z +0.000,A -0.000,E1 -46.493,E3 +78911.263,E4 +0.000} C_DIS
LIN {X -190.174,Y +1086.028,Z +0.000,A -0.000,E1 -46.483,E3 +78920.157,E4 +0.000} C_DIS
LIN {X -190.200,Y +1096.186,Z +0.000,A -0.000,E1 -46.448,E3 +78933.161,E4 +0.000} C_DIS
LIN {X -190.154,Y +1108.998,Z +0.000,A -0.054,E1 -46.295,E3 +78949.656,E4 +0.000} C_DIS
LIN {X -189.772,Y +1119.341,Z +0.000,A -0.752,E1 -45.902,E3 +78963.194,E4 +0.000} C_DIS
LIN {X -189.097,Y +1124.276,Z +0.000,A -2.508,E1 -45.397,E3 +78969.926,E4 +0.000} C_DIS
LIN {X -187.410,Y +1129.069,Z +0.000,A -5.304,E1 -44.585,E3 +78977.099,E4 +0.000} C_DIS
LIN {X -183.899,Y +1134.873,Z +0.000,A -10.372,E1 -42.805,E3 +78987.105,E4 +0.000} C_DIS
LIN {X -179.711,Y +1140.065,Z +0.000,A -15.940,E1 -40.393,E3 +78997.891,E4 +0.000} C_DIS
LIN {X -176.763,Y +1143.197,Z +0.000,A -18.748,E1 -38.674,E3 +79005.629,E4 +0.000} C_DIS
LIN {X -172.185,Y +1147.423,Z +0.000,A -19.971,E1 -36.175,E3 +79018.359,E4 +0.000} C_DIS
LIN {X -165.999,Y +1152.127,Z +0.000,A -20.000,E1 -32.027,E3 +79038.117,E4 +0.000} C_DIS
LIN {X -160.138,Y +1155.667,Z +0.000,A -20.000,E1 -26.368,E3 +79062.487,E4 +0.000} C_DIS
LIN {X -155.625,Y +1157.756,Z +0.000,A -20.000,E1 -19.505,E3 +79091.163,E4 +0.000} C_DIS
LIN {X -153.552,Y +1158.113,Z +0.000,A -20.000,E1 -11.113,E3 +79126.914,E4 +0.000} C_DIS
LIN {X -156.311,Y +1155.540,Z +0.000,A -20.000,E1 -0.839,E3 +79170.274,E4 +0.000} C_DIS
LIN {X -161.281,Y +1151.851,Z +0.000,A -20.000,E1 +7.737,E3 +79200.173,E4 +0.000} C_DIS
LIN {X -167.493,Y +1147.157,Z +0.000,A -20.000,E1 +16.195,E3 +79224.612,E4 +0.000} C_DIS
LIN {X -173.235,Y +1142.221,Z +0.000,A -20.000,E1 +22.930,E3 +79241.914,E4 +0.000} C_DIS
LIN {X -181.123,Y +1133.734,Z +0.000,A -20.000,E1 +30.868,E3 +79262.670,E4 +0.000} C_DIS
LIN {X -189.654,Y +1120.856,Z +0.000,A -20.000,E1 +39.018,E3 +79284.684,E4 +0.000} C_DIS
LIN {X -195.246,Y +1107.046,Z +0.000,A -20.000,E1 +44.515,E3 +79302.586,E4 +0.000} C_DIS
LIN {X -198.051,Y +1092.368,Z +0.000,A -20.000,E1 +47.947,E3 +79319.112,E4 +0.000} C_DIS
LIN {X -198.143,Y +1081.370,Z +0.000,A -19.806,E1 +49.153,E3 +79330.973,E4 +0.000} C_DIS
LIN {X -197.177,Y +1073.569,Z +0.000,A -17.356,E1 +49.162,E3 +79339.557,E4 +0.000} C_DIS
LIN {X -195.448,Y +1066.139,Z +0.000,A -12.154,E1 +48.512,E3 +79348.152,E4 +0.000} C_DIS
LIN {X -193.346,Y +1058.941,Z +0.000,A -7.133,E1 +47.724,E3 +79357.032,E4 +0.000} C_DIS
LIN {X -191.781,Y +1050.839,Z +0.000,A -3.715,E1 +47.274,E3 +79367.365,E4 +0.000} C_DIS
LIN {X -190.795,Y +1039.355,Z +0.000,A -0.983,E1 +46.842,E3 +79382.025,E4 +0.000} C_DIS
LIN {X -190.395,Y +1028.856,Z +0.000,A -0.089,E1 +46.598,E3 +79395.419,E4 +0.000} C_DIS
LIN {X -190.239,Y +1018.851,Z +0.000,A -0.004,E1 +46.529,E3 +79408.187,E4 +0.000} C_DIS
LIN {X -190.161,Y +1004.975,Z +0.000,A +0.000,E1 +46.506,E3 +79425.901,E4 +0.000} C_DIS
LIN {X -190.142,Y +412.853,Z +0.000,A +0.000,E1 +46.501,E3 +80182.107,E4 +0.000} C_DIS
LIN {X -190.147,Y +401.077,Z +0.000,A +0.000,E1 +46.499,E3 +80197.148,E4 +0.000} C_DIS
LIN {X -190.159,Y +390.929,Z +0.000,A +0.000,E1 +46.494,E3 +80210.114,E4 +0.000} C_DIS
LIN {X -190.174,Y +383.973,Z +0.000,A +0.000,E1 +46.484,E3 +80219.007,E4 +0.000} C_DIS
LIN {X -190.200,Y +373.815,Z +0.000,A +0.000,E1 +46.448,E3 +80232.012,E4 +0.000} C_DIS
LIN {X -190.154,Y +361.003,Z +0.000,A +0.000,E1 +46.303,E3 +80248.506,E4 +0.000} C_DIS
LIN {X -189.772,Y +350.660,Z +0.000,A +0.049,E1 +45.996,E3 +80262.045,E4 +0.000} C_DIS
LIN {X -189.325,Y +346.917,Z +0.000,A +0.243,E1 +45.771,E3 +80267.114,E4 +0.000} C_DIS
LIN {X -188.196,Y +342.754,Z +0.000,A +1.966,E1 +45.249,E3 +80273.122,E4 +0.000} C_DIS
LIN {X -185.199,Y +337.023,Z +0.000,A +6.630,E1 +43.793,E3 +80282.496,E4 +0.000} C_DIS
LIN {X -181.141,Y +331.596,Z +0.000,A +12.274,E1 +41.569,E3 +80293.056,E4 +0.000} C_DIS
LIN {X -176.762,Y +326.804,Z +0.000,A +17.560,E1 +38.898,E3 +80304.480,E4 +0.000} C_DIS
LIN {X -172.184,Y +322.578,Z +0.000,A +19.859,E1 +36.197,E3 +80317.210,E4 +0.000} C_DIS
LIN {X -165.998,Y +317.874,Z +0.000,A +20.000,E1 +32.027,E3 +80336.968,E4 +0.000} C_DIS
LIN {X -160.137,Y +314.334,Z +0.000,A +20.000,E1 +26.368,E3 +80361.337,E4 +0.000} C_DIS
LIN {X -155.624,Y +312.245,Z +0.000,A +20.000,E1 +19.506,E3 +80390.013,E4 +0.000} C_DIS
LIN {X -153.557,Y +311.879,Z +0.000,A +20.000,E1 +11.113,E3 +80425.768,E4 +0.000} C_DIS
LIN {X -155.320,Y +313.348,Z +0.000,A +20.000,E1 +3.401,E3 +80458.952,E4 +0.000} C_DIS
LIN {X -160.005,Y +315.804,Z +0.000,A +20.000,E1 -4.720,E3 +80489.330,E4 +0.000} C_DIS
LIN {X -164.504,Y +318.255,Z +0.000,A +20.000,E1 -10.663,E3 +80508.699,E4 +0.000} C_DIS
LIN {X -170.340,Y +322.684,Z +0.000,A +20.000,E1 -17.457,E3 +80528.731,E4 +0.000} C_DIS
LIN {X -175.568,Y +329.106,Z +0.000,A +20.000,E1 -24.747,E3 +80545.965,E4 +0.000} C_DIS
LIN {X -184.074,Y +340.065,Z +0.000,A +20.000,E1 -33.664,E3 +80568.905,E4 +0.000} C_DIS
LIN {X -190.779,Y +351.388,Z +0.000,A +20.000,E1 -40.083,E3 +80586.683,E4 +0.000} C_DIS
LIN {X -195.254,Y +362.955,Z +0.000,A +20.000,E1 -44.515,E3 +80601.436,E4 +0.000} C_DIS
LIN {X -197.754,Y +374.780,Z +0.000,A +20.000,E1 -47.450,E3 +80614.858,E4 +0.000} C_DIS
LIN {X -198.310,Y +383.215,Z +0.000,A +19.956,E1 -48.698,E3 +80623.982,E4 +0.000} C_DIS
LIN {X -197.912,Y +391.275,Z +0.000,A +18.601,E1 -49.158,E3 +80632.700,E4 +0.000} C_DIS
LIN {X -196.679,Y +398.944,Z +0.000,A +13.989,E1 -48.784,E3 +80641.254,E4 +0.000} C_DIS
LIN {X -194.742,Y +406.288,Z +0.000,A +8.476,E1 -48.001,E3 +80649.937,E4 +0.000} C_DIS
LIN {X -192.748,Y +413.472,Z +0.000,A +3.905,E1 -47.267,E3 +80658.947,E4 +0.000} C_DIS
LIN {X -191.781,Y +419.162,Z +0.000,A +1.739,E1 -46.975,E3 +80666.215,E4 +0.000} C_DIS
LIN {X -190.795,Y +430.646,Z +0.000,A +0.152,E1 -46.707,E3 +80680.876,E4 +0.000} C_DIS
LIN {X -190.395,Y +441.145,Z +0.000,A +0.001,E1 -46.583,E3 +80694.269,E4 +0.000} C_DIS
LIN {X -190.239,Y +451.150,Z +0.000,A -0.000,E1 -46.528,E3 +80707.037,E4 +0.000} C_DIS
LIN {X -190.161,Y +465.026,Z +0.000,A -0.000,E1 -46.506,E3 +80724.752,E4 +0.000} C_DIS
LIN {X -190.142,Y +1057.148,Z +0.000,A -0.000,E1 -46.500,E3 +81480.958,E4 +0.000} C_DIS
LIN {X -190.147,Y +1068.924,Z +0.000,A -0.000,E1 -46.499,E3 +81495.999,E4 +0.000} C_DIS
LIN {X -190.159,Y +1079.072,Z +0.000,A -0.000,E1 -46.493,E3 +81508.964,E4 +0.000} C_DIS
LIN {X -190.174,Y +1086.028,Z +0.000,A -0.000,E1 -46.483,E3 +81517.858,E4 +0.000} C_DIS
LIN {X -190.200,Y +1096.186,Z +0.000,A -0.000,E1 -46.448,E3 +81530.862,E4 +0.000} C_DIS
LIN {X -190.154,Y +1108.998,Z +0.000,A -0.054,E1 -46.295,E3 +81547.357,E4 +0.000} C_DIS
LIN {X -189.772,Y +1119.341,Z +0.000,A -0.752,E1 -45.902,E3 +81560.895,E4 +0.000} C_DIS
LIN {X -189.097,Y +1124.276,Z +0.000,A -2.508,E1 -45.397,E3 +81567.627,E4 +0.000} C_DIS
LIN {X -187.410,Y +1129.069,Z +0.000,A -5.304,E1 -44.585,E3 +81574.800,E4 +0.000} C_DIS
LIN {X -183.899,Y +1134.873,Z +0.000,A -10.372,E1 -42.805,E3 +81584.806,E4 +0.000} C_DIS
LIN {X -179.711,Y +1140.065,Z +0.000,A -15.940,E1 -40.393,E3 +81595.592,E4 +0.000} C_DIS
LIN {X -176.763,Y +1143.197,Z +0.000,A -18.748,E1 -38.674,E3 +81603.330,E4 +0.000} C_DIS
LIN {X -172.185,Y +1147.423,Z +0.000,A -19.971,E1 -36.175,E3 +81616.060,E4 +0.000} C_DIS
LIN {X -165.999,Y +1152.127,Z +0.000,A -20.000,E1 -32.027,E3 +81635.818,E4 +0.000} C_DIS
LIN {X -160.138,Y +1155.667,Z +0.000,A -20.000,E1 -26.368,E3 +81660.188,E4 +0.000} C_DIS
LIN {X -155.625,Y +1157.756,Z +0.000,A -20.000,E1 -19.505,E3 +81688.864,E4 +0.000} C_DIS
LIN {X -153.552,Y +1158.113,Z +0.000,A -20.000,E1 -11.113,E3 +81724.615,E4 +0.000} C_DIS
LIN {X -156.311,Y +1155.540,Z +0.000,A -20.000,E1 -0.839,E3 +81767.975,E4 +0.000} C_DIS
LIN {X -161.281,Y +1151.851,Z +0.000,A -20.000,E1 +7.737,E3 +81797.874,E4 +0.000} C_DIS
LIN {X -167.493,Y +1147.157,Z +0.000,A -20.000,E1 +16.195,E3 +81822.313,E4 +0.000} C_DIS
LIN {X -173.235,Y +1142.221,Z +0.000,A -20.000,E1 +22.930,E3 +81839.615,E4 +0.000} C_DIS
LIN {X -181.123,Y +1133.734,Z +0.000,A -20.000,E1 +30.868,E3 +81860.371,E4 +0.000} C_DIS
LIN {X -189.654,Y +1120.856,Z +0.000,A -20.000,E1 +39.018,E3 +81882.385,E4 +0.000} C_DIS
LIN {X -195.246,Y +1107.046,Z +0.000,A -20.000,E1 +44.515,E3 +81900.287,E4 +0.000} C_DIS
LIN {X -198.051,Y +1092.368,Z +0.000,A -20.000,E1 +47.947,E3 +81916.813,E4 +0.000} C_DIS
LIN {X -198.143,Y +1081.370,Z +0.000,A -19.806,E1 +49.153,E3 +81928.674,E4 +0.000} C_DIS
LIN {X -197.177,Y +1073.569,Z +0.000,A -17.356,E1 +49.162,E3 +81937.258,E4 +0.000} C_DIS
LIN {X -195.448,Y +1066.139,Z +0.000,A -12.154,E1 +48.512,E3 +81945.853,E4 +0.000} C_DIS
LIN {X -193.346,Y +1058.941,Z +0.000,A -7.133,E1 +47.724,E3 +81954.733,E4 +0.000} C_DIS
LIN {X -191.781,Y +1050.839,Z +0.000,A -3.715,E1 +47.274,E3 +81965.066,E4 +0.000} C_DIS
LIN {X -190.795,Y +1039.355,Z +0.000,A -0.983,E1 +46.842,E3 +81979.726,E4 +0.000} C_DIS
LIN {X -190.395,Y +1028.856,Z +0.000,A -0.089,E1 +46.598,E3 +81993.120,E4 +0.000} C_DIS
LIN {X -190.239,Y +1018.851,Z +0.000,A -0.004,E1 +46.529,E3 +82005.888,E4 +0.000} C_DIS
LIN {X -190.161,Y +1004.975,Z +0.000,A +0.000,E1 +46.506,E3 +82023.602,E4 +0.000} C_DIS
LIN {X -190.142,Y +412.853,Z +0.000,A +0.000,E1 +46.501,E3 +82779.808,E4 +0.000} C_DIS
LIN {X -190.147,Y +401.077,Z +0.000,A +0.000,E1 +46.499,E3 +82794.849,E4 +0.000} C_DIS
LIN {X -190.159,Y +390.929,Z +0.000,A +0.000,E1 +46.494,E3 +82807.815,E4 +0.000} C_DIS
LIN {X -190.174,Y +383.973,Z +0.000,A +0.000,E1 +46.484,E3 +82816.708,E4 +0.000} C_DIS
LIN {X -190.200,Y +373.815,Z +0.000,A +0.000,E1 +46.448,E3 +82829.713,E4 +0.000} C_DIS
LIN {X -190.154,Y +361.003,Z +0.000,A +0.000,E1 +46.303,E3 +82846.207,E4 +0.000} C_DIS
LIN {X -189.772,Y +350.660,Z +0.000,A +0.049,E1 +45.996,E3 +82859.746,E4 +0.000} C_DIS
LIN {X -189.325,Y +346.917,Z +0.000,A +0.243,E1 +45.771,E3 +82864.815,E4 +0.000} C_DIS
LIN {X -188.196,Y +342.754,Z +0.000,A +1.966,E1 +45.249,E3 +82870.823,E4 +0.000} C_DIS
LIN {X -185.199,Y +337.023,Z +0.000,A +6.630,E1 +43.793,E3 +82880.197,E4 +0.000} C_DIS
LIN {X -181.141,Y +331.596,Z +0.000,A +12.274,E1 +41.569,E3 +82890.757,E4 +0.000} C_DIS
LIN {X -176.762,Y +326.804,Z +0.000,A +17.560,E1 +38.898,E3 +82902.181,E4 +0.000} C_DIS
LIN {X -172.184,Y +322.578,Z +0.000,A +19.859,E1 +36.197,E3 +82914.911,E4 +0.000} C_DIS
LIN {X -165.998,Y +317.874,Z +0.000,A +20.000,E1 +32.027,E3 +82934.669,E4 +0.000} C_DIS
LIN {X -160.137,Y +314.334,Z +0.000,A +20.000,E1 +26.368,E3 +82959.038,E4 +0.000} C_DIS
LIN {X -155.624,Y +312.245,Z +0.000,A +20.000,E1 +19.506,E3 +82987.714,E4 +0.000} C_DIS
LIN {X -153.557,Y +311.879,Z +0.000,A +20.000,E1 +11.113,E3 +83023.469,E4 +0.000} C_DIS
LIN {X -155.320,Y +313.348,Z +0.000,A +20.000,E1 +3.401,E3 +83056.653,E4 +0.000} C_DIS
LIN {X -160.005,Y +315.804,Z +0.000,A +20.000,E1 -4.720,E3 +83087.031,E4 +0.000} C_DIS
LIN {X -164.504,Y +318.255,Z +0.000,A +20.000,E1 -10.663,E3 +83106.400,E4 +0.000} C_DIS
LIN {X -170.340,Y +322.684,Z +0.000,A +20.000,E1 -17.457,E3 +83126.432,E4 +0.000} C_DIS
LIN {X -175.568,Y +329.106,Z +0.000,A +20.000,E1 -24.747,E3 +83143.666,E4 +0.000} C_DIS
LIN {X -184.074,Y +340.065,Z +0.000,A +20.000,E1 -33.664,E3 +83166.606,E4 +0.000} C_DIS
LIN {X -190.779,Y +351.388,Z +0.000,A +20.000,E1 -40.083,E3 +83184.384,E4 +0.000} C_DIS
LIN {X -195.254,Y +362.955,Z +0.000,A +20.000,E1 -44.515,E3 +83199.137,E4 +0.000} C_DIS
LIN {X -197.754,Y +374.780,Z +0.000,A +20.000,E1 -47.450,E3 +83212.559,E4 +0.000} C_DIS
LIN {X -198.310,Y +383.215,Z +0.000,A +19.956,E1 -48.698,E3 +83221.683,E4 +0.000} C_DIS
LIN {X -197.912,Y +391.275,Z +0.000,A +18.601,E1 -49.158,E3 +83230.401,E4 +0.000} C_DIS
LIN {X -196.679,Y +398.944,Z +0.000,A +13.989,E1 -48.784,E3 +83238.955,E4 +0.000} C_DIS
LIN {X -194.742,Y +406.288,Z +0.000,A +8.476,E1 -48.001,E3 +83247.638,E4 +0.000} C_DIS
LIN {X -192.748,Y +413.472,Z +0.000,A +3.905,E1 -47.267,E3 +83256.648,E4 +0.000} C_DIS
LIN {X -191.781,Y +419.162,Z +0.000,A +1.739,E1 -46.975,E3 +83263.916,E4 +0.000} C_DIS
LIN {X -190.795,Y +430.646,Z +0.000,A +0.152,E1 -46.707,E3 +83278.577,E4 +0.000} C_DIS
LIN {X -190.395,Y +441.145,Z +0.000,A +0.001,E1 -46.583,E3 +83291.970,E4 +0.000} C_DIS
LIN {X -190.239,Y +451.150,Z +0.000,A -0.000,E1 -46.528,E3 +83304.738,E4 +0.000} C_DIS
LIN {X -190.161,Y +465.026,Z +0.000,A -0.000,E1 -46.506,E3 +83322.453,E4 +0.000} C_DIS
LIN {X -190.142,Y +1057.148,Z +0.000,A -0.000,E1 -46.500,E3 +84078.659,E4 +0.000} C_DIS
LIN {X -190.147,Y +1068.924,Z +0.000,A -0.000,E1 -46.499,E3 +84093.700,E4 +0.000} C_DIS
LIN {X -190.159,Y +1079.072,Z +0.000,A -0.000,E1 -46.493,E3 +84106.665,E4 +0.000} C_DIS
LIN {X -190.174,Y +1086.028,Z +0.000,A -0.000,E1 -46.483,E3 +84115.559,E4 +0.000} C_DIS
LIN {X -190.200,Y +1096.186,Z +0.000,A -0.000,E1 -46.448,E3 +84128.563,E4 +0.000} C_DIS
LIN {X -190.154,Y +1108.998,Z +0.000,A -0.054,E1 -46.295,E3 +84145.058,E4 +0.000} C_DIS
LIN {X -189.772,Y +1119.341,Z +0.000,A -0.752,E1 -45.902,E3 +84158.596,E4 +0.000} C_DIS
LIN {X -189.097,Y +1124.276,Z +0.000,A -2.508,E1 -45.397,E3 +84165.328,E4 +0.000} C_DIS
LIN {X -187.410,Y +1129.069,Z +0.000,A -5.304,E1 -44.585,E3 +84172.501,E4 +0.000} C_DIS
LIN {X -183.899,Y +1134.873,Z +0.000,A -10.372,E1 -42.805,E3 +84182.507,E4 +0.000} C_DIS
LIN {X -179.711,Y +1140.065,Z +0.000,A -15.940,E1 -40.393,E3 +84193.293,E4 +0.000} C_DIS
LIN {X -176.763,Y +1143.197,Z +0.000,A -18.748,E1 -38.674,E3 +84201.031,E4 +0.000} C_DIS
